LIN {X 0,Y 368.929,Z 1065.584,A -85,B 0,C 180,E1 16268.801,E2 16268.801} C_VEL
LIN {X 0,Y 361.367,Z 1080.301,A -85,B 0,C 180,E1 16265.652,E2 16265.652} C_VEL
LIN {X 0,Y 353.629,Z 1094.954,A -85,B 0,C 180,E1 16261.908,E2 16261.908} C_VEL
LIN {X 0,Y 348.28,Z 1105.205,A -85,B 0,C 180,E1 16258.82,E2 16258.82} C_VEL
LIN {X 0,Y 344.292,Z 1113.061,A -85,B 0,C 180,E1 16256.113,E2 16256.113} C_VEL
LIN {X 0,Y 341.847,Z 1116.356,A -85,B 0,C 180,E1 16255.008,E2 16255.008} C_VEL
LIN {X 0,Y 332.302,Z 1125.106,A -85,B 0,C 180,E1 16252.144,E2 16252.144} C_VEL
LIN {X 0,Y 330.487,Z 1127.448,A -85,B 0,C 180,E1 16251.111,E2 16251.111} C_VEL
LIN {X 0,Y 327.162,Z 1134.807,A -85,B 0,C 180,E1 16247.181,E2 16247.181} C_VEL
LIN {X 0,Y 324.967,Z 1140.258,A -85,B 0,C 180,E1 16243.693,E2 16243.693} C_VEL
LIN {X 0,Y 323.573,Z 1144.448,A -85,B 0,C 180,E1 16240.461,E2 16240.461} C_VEL
LIN {X 0,Y 322.533,Z 1148.193,A -85,B 0,C 180,E1 16236.887,E2 16236.887} C_VEL
LIN {X 0,Y 321.986,Z 1150.9,A -85,B 0,C 180,E1 16233.557,E2 16233.557} C_VEL
LIN {X 0,Y 321.773,Z 1152.88,A -85,B 0,C 180,E1 16230.226,E2 16230.226} C_VEL
LIN {X 0,Y 321.676,Z 1154.208,A -85,B 0,C 180,E1 16226.79,E2 16226.79} C_VEL
LIN {X 0,Y 321.778,Z 1154.811,A -85,B 0,C 180,E1 16223.438,E2 16223.438} C_VEL
LIN {X 0,Y 322.051,Z 1154.692,A -85,B 0,C 180,E1 16219.827,E2 16219.827} C_VEL
LIN {X 0,Y 322.549,Z 1153.785,A -85,B 0,C 180,E1 16216.2,E2 16216.2} C_VEL
LIN {X 0,Y 323.386,Z 1152.158,A -85,B 0,C 180,E1 16212.681,E2 16212.681} C_VEL
LIN {X 0,Y 324.964,Z 1149.492,A -85,B 0,C 180,E1 16208.85,E2 16208.85} C_VEL
LIN {X 0,Y 327.742,Z 1145.238,A -85,B 0,C 180,E1 16204.374,E2 16204.374} C_VEL
LIN {X 0,Y 332.024,Z 1139.047,A -85,B 0,C 180,E1 16199.655,E2 16199.655} C_VEL
LIN {X 0,Y 336.888,Z 1132.582,A -85,B 0,C 180,E1 16195.74,E2 16195.74} C_VEL
LIN {X 0,Y 344.034,Z 1123.589,A -85,B 0,C 180,E1 16191.307,E2 16191.307} C_VEL
LIN {X 0,Y 351.989,Z 1113.581,A -85,B 0,C 180,E1 16187.365,E2 16187.365} C_VEL
LIN {X 0,Y 361.723,Z 1101.762,A -85,B 0,C 180,E1 16183.458,E2 16183.458} C_VEL
LIN {X 0,Y 372.861,Z 1088.013,A -85,B 0,C 180,E1 16179.761,E2 16179.761} C_VEL
LIN {X 0,Y 385.536,Z 1072.73,A -85,B 0,C 180,E1 16176.297,E2 16176.297} C_VEL
LIN {X 0,Y 402.18,Z 1053.149,A -85,B 0,C 180,E1 16172.616,E2 16172.616} C_VEL
LIN {X 0,Y 414.234,Z 1039.577,A -85,B 0,C 180,E1 16170.456,E2 16170.456} C_VEL
LIN {X 0,Y 397.297,Z 1065.107,A -85,B 0,C 180,E1 16167.737,E2 16167.737} C_VEL
LIN {X 0,Y 379.335,Z 1097.703,A -85,B 0,C 180,E1 16163.762,E2 16163.762} C_VEL
LIN {X 0,Y 366.086,Z 1125.2,A -85,B 0,C 180,E1 16159.865,E2 16159.865} C_VEL
LIN {X 0,Y 355.502,Z 1148.51,A -85,B 0,C 180,E1 16155.995,E2 16155.995} C_VEL
LIN {X 0,Y 348.419,Z 1164.919,A -85,B 0,C 180,E1 16152.854,E2 16152.854} C_VEL
LIN {X 0,Y 342.515,Z 1179.307,A -85,B 0,C 180,E1 16149.74,E2 16149.74} C_VEL
LIN {X 0,Y 337.4,Z 1192.323,A -85,B 0,C 180,E1 16146.559,E2 16146.559} C_VEL
LIN {X 0,Y 333.277,Z 1203.483,A -85,B 0,C 180,E1 16143.483,E2 16143.483} C_VEL
LIN {X 0,Y 329.754,Z 1213.978,A -85,B 0,C 180,E1 16140.21,E2 16140.21} C_VEL
LIN {X 0,Y 326.806,Z 1223.77,A -85,B 0,C 180,E1 16136.728,E2 16136.728} C_VEL
LIN {X 0,Y 324.695,Z 1231.919,A -85,B 0,C 180,E1 16133.406,E2 16133.406} C_VEL
LIN {X 0,Y 323.147,Z 1239.311,A -85,B 0,C 180,E1 16129.899,E2 16129.899} C_VEL
LIN {X 0,Y 322.162,Z 1245.863,A -85,B 0,C 180,E1 16126.22,E2 16126.22} C_VEL
LIN {X 0,Y 321.683,Z 1251.131,A -85,B 0,C 180,E1 16122.567,E2 16122.567} C_VEL
LIN {X 0,Y 321.55,Z 1254.796,A -85,B 0,C 180,E1 16119.305,E2 16119.305} C_VEL
LIN {X 0,Y 321.644,Z 1257.645,A -85,B 0,C 180,E1 16115.855,E2 16115.855} C_VEL
LIN {X 0,Y 321.714,Z 1259.335,A -85,B 0,C 180,E1 16112.494,E2 16112.494} C_VEL
LIN {X 0,Y 321.649,Z 1259.923,A -85,B 0,C 180,E1 16109.109,E2 16109.109} C_VEL
LIN {X 0,Y 321.554,Z 1259.487,A -85,B 0,C 180,E1 16105.899,E2 16105.899} C_VEL
LIN {X 0,Y 321.358,Z 1257.951,A -85,B 0,C 180,E1 16102.491,E2 16102.491} C_VEL
LIN {X 0,Y 321.322,Z 1255.176,A -85,B 0,C 180,E1 16098.876,E2 16098.876} C_VEL
LIN {X 0,Y 321.576,Z 1251.22,A -85,B 0,C 180,E1 16095.229,E2 16095.229} C_VEL
LIN {X 0,Y 322.325,Z 1246.263,A -85,B 0,C 180,E1 16091.669,E2 16091.669} C_VEL
LIN {X 0,Y 323.717,Z 1240.102,A -85,B 0,C 180,E1 16088.054,E2 16088.054} C_VEL
LIN {X 0,Y 325.87,Z 1232.599,A -85,B 0,C 180,E1 16084.365,E2 16084.365} C_VEL
LIN {X 0,Y 329.419,Z 1222.452,A -85,B 0,C 180,E1 16080.146,E2 16080.146} C_VEL
LIN {X 0,Y 334.451,Z 1209.771,A -85,B 0,C 180,E1 16075.803,E2 16075.803} C_VEL
LIN {X 0,Y 339.559,Z 1198.071,A -85,B 0,C 180,E1 16072.384,E2 16072.384} C_VEL
LIN {X 0,Y 345.401,Z 1185.305,A -85,B 0,C 180,E1 16069.139,E2 16069.139} C_VEL
LIN {X 0,Y 353.389,Z 1168.407,A -85,B 0,C 180,E1 16065.437,E2 16065.437} C_VEL
LIN {X 0,Y 361.45,Z 1151.342,A -85,B 0,C 180,E1 16062.304,E2 16062.304} C_VEL
LIN {X 0,Y 369.122,Z 1135.016,A -85,B 0,C 180,E1 16059.709,E2 16059.709} C_VEL
LIN {X 0,Y 377.835,Z 1116.171,A -85,B 0,C 180,E1 16057.112,E2 16057.112} C_VEL
LIN {X 0,Y 387.715,Z 1093.832,A -85,B 0,C 180,E1 16054.517,E2 16054.517} C_VEL
LIN {X 0,Y 395.54,Z 1075.271,A -85,B 0,C 180,E1 16052.671,E2 16052.671} C_VEL
LIN {X 0,Y 403.455,Z 1055.515,A -85,B 0,C 180,E1 16050.964,E2 16050.964} C_VEL
LIN {X 0,Y 412.389,Z 1031.699,A -85,B 0,C 180,E1 16049.208,E2 16049.208} C_VEL
LIN {X 0,Y 420.728,Z 1007.097,A -85,B 0,C 180,E1 16047.716,E2 16047.716} C_VEL
LIN {X 0,Y 427.295,Z 986.002,A -85,B 0,C 180,E1 16046.634,E2 16046.634} C_VEL
LIN {X 0,Y 434.084,Z 962.064,A -85,B 0,C 180,E1 16045.606,E2 16045.606} C_VEL
LIN {X 0,Y 440.942,Z 933.969,A -85,B 0,C 180,E1 16044.644,E2 16044.644} C_VEL
LIN {X 0,Y 445.717,Z 910.846,A -85,B 0,C 180,E1 16044.015,E2 16044.015} C_VEL
LIN {X 0,Y 449.567,Z 887.226,A -85,B 0,C 180,E1 16043.462,E2 16043.462} C_VEL
LIN {X 0,Y 453.668,Z 850.311,A -85,B 0,C 180,E1 16042.756,E2 16042.756} C_VEL
LIN {X 0,Y 474.582,Z 637.863,A -85,B 0,C 180,E1 16039.052,E2 16039.052} C_VEL
LIN {X 0,Y 480.593,Z 579.148,A -85,B 0,C 180,E1 16038.031,E2 16038.031} C_VEL
LIN {X 0,Y 471.163,Z 563.283,A -85,B 0,C 180,E1 16034.942,E2 16034.942} C_VEL
LIN {X 0,Y 462.699,Z 549.888,A -85,B 0,C 180,E1 16031.878,E2 16031.878} C_VEL
LIN {X 0,Y 454.912,Z 537.8,A -85,B 0,C 180,E1 16028.723,E2 16028.723} C_VEL
LIN {X 0,Y 448.462,Z 528.192,A -85,B 0,C 180,E1 16025.822,E2 16025.822} C_VEL
LIN {X 0,Y 442.933,Z 519.88,A -85,B 0,C 180,E1 16023.041,E2 16023.041} C_VEL
LIN {X 0,Y 437.602,Z 512.312,A -85,B 0,C 180,E1 16020.065,E2 16020.065} C_VEL
LIN {X 0,Y 434.436,Z 507.764,A -85,B 0,C 180,E1 16018.087,E2 16018.087} C_VEL
LIN {X 0,Y 431.277,Z 503.161,A -85,B 0,C 180,E1 16015.945,E2 16015.945} C_VEL
LIN {X 0,Y 428.043,Z 498.552,A -85,B 0,C 180,E1 16013.562,E2 16013.562} C_VEL
LIN {X 0,Y 424.911,Z 493.865,A -85,B 0,C 180,E1 16010.929,E2 16010.929} C_VEL
LIN {X 0,Y 421.631,Z 489.288,A -85,B 0,C 180,E1 16007.815,E2 16007.815} C_VEL
LIN {X 0,Y 420.488,Z 487.518,A -85,B 0,C 180,E1 16006.546,E2 16006.546} C_VEL
LIN {X 0,Y 417.521,Z 483.166,A -85,B 0,C 180,E1 16002.868,E2 16002.868} C_VEL
LIN {X 0,Y 414.516,Z 480.784,A -85,B 0,C 180,E1 15998.787,E2 15998.787} C_VEL
LIN {X 0,Y 412.902,Z 477.95,A -85,B 0,C 180,E1 15995.385,E2 15995.385} C_VEL
LIN {X 0,Y 412.303,Z 476.965,A -85,B 0,C 180,E1 15993.653,E2 15993.653} C_VEL
LIN {X 0,Y 410.774,Z 476.217,A -85,B 0,C 180,E1 15989.095,E2 15989.095} C_VEL
LIN {X 0,Y 410.291,Z 475.897,A -85,B 0,C 180,E1 15985.212,E2 15985.212} C_VEL
LIN {X 0,Y 410.589,Z 476.045,A -85,B 0,C 180,E1 15980.531,E2 15980.531} C_VEL
LIN {X 0,Y 411.65,Z 476.625,A -85,B 0,C 180,E1 15976.371,E2 15976.371} C_VEL
LIN {X 0,Y 412.909,Z 477.464,A -85,B 0,C 180,E1 15973.408,E2 15973.408} C_VEL
LIN {X 0,Y 414.387,Z 480.345,A -85,B 0,C 180,E1 15970.29,E2 15970.29} C_VEL
LIN {X 0,Y 417.361,Z 482.989,A -85,B 0,C 180,E1 15966.281,E2 15966.281} C_VEL
LIN {X 0,Y 418.392,Z 483.769,A -85,B 0,C 180,E1 15965.166,E2 15965.166} C_VEL
LIN {X 0,Y 421.167,Z 487.9,A -85,B 0,C 180,E1 15962.126,E2 15962.126} C_VEL
LIN {X 0,Y 423.64,Z 489.996,A -85,B 0,C 180,E1 15959.979,E2 15959.979} C_VEL
LIN {X 0,Y 426.809,Z 494.304,A -85,B 0,C 180,E1 15957.39,E2 15957.39} C_VEL
LIN {X 0,Y 428.742,Z 496.203,A -85,B 0,C 180,E1 15956.05,E2 15956.05} C_VEL
LIN {X 0,Y 432.452,Z 500.769,A -85,B 0,C 180,E1 15953.578,E2 15953.578} C_VEL
LIN {X 0,Y 433.913,Z 502.443,A -85,B 0,C 180,E1 15952.704,E2 15952.704} C_VEL
LIN {X 0,Y 438.68,Z 508.376,A -85,B 0,C 180,E1 15949.992,E2 15949.992} C_VEL
LIN {X 0,Y 443.421,Z 514.255,A -85,B 0,C 180,E1 15947.587,E2 15947.587} C_VEL
LIN {X 0,Y 447.969,Z 520.088,A -85,B 0,C 180,E1 15945.47,E2 15945.47} C_VEL
LIN {X 0,Y 454.659,Z 528.643,A -85,B 0,C 180,E1 15942.669,E2 15942.669} C_VEL
LIN {X 0,Y 463.73,Z 540.901,A -85,B 0,C 180,E1 15939.272,E2 15939.272} C_VEL
LIN {X 0,Y 474.803,Z 556.321,A -85,B 0,C 180,E1 15935.65,E2 15935.65} C_VEL
LIN {X 0,Y 476.31,Z 558.799,A -85,B 0,C 180,E1 15935.176,E2 15935.176} C_VEL
LIN {X 0,Y 455.359,Z 771.033,A -85,B 0,C 180,E1 15931.537,E2 15931.537} C_VEL
LIN {X 0,Y 451.923,Z 800.539,A -85,B 0,C 180,E1 15930.948,E2 15930.948} C_VEL
LIN {X 0,Y 448.327,Z 824.07,A -85,B 0,C 180,E1 15930.335,E2 15930.335} C_VEL
LIN {X 0,Y 443.229,Z 851.426,A -85,B 0,C 180,E1 15929.441,E2 15929.441} C_VEL
LIN {X 0,Y 437.133,Z 877.659,A -85,B 0,C 180,E1 15928.362,E2 15928.362} C_VEL
LIN {X 0,Y 431.224,Z 899.891,A -85,B 0,C 180,E1 15927.276,E2 15927.276} C_VEL
LIN {X 0,Y 423.599,Z 925.285,A -85,B 0,C 180,E1 15925.804,E2 15925.804} C_VEL
LIN {X 0,Y 415.695,Z 948.263,A -85,B 0,C 180,E1 15924.202,E2 15924.202} C_VEL
LIN {X 0,Y 408.347,Z 967.91,A -85,B 0,C 180,E1 15922.613,E2 15922.613} C_VEL
LIN {X 0,Y 399.847,Z 988.995,A -85,B 0,C 180,E1 15920.646,E2 15920.646} C_VEL
LIN {X 0,Y 390.613,Z 1009.923,A -85,B 0,C 180,E1 15918.333,E2 15918.333} C_VEL
LIN {X 0,Y 382.76,Z 1026.711,A -85,B 0,C 180,E1 15916.179,E2 15916.179} C_VEL
LIN {X 0,Y 375.211,Z 1042.141,A -85,B 0,C 180,E1 15913.91,E2 15913.91} C_VEL
LIN {X 0,Y 366.367,Z 1059.568,A -85,B 0,C 180,E1 15910.943,E2 15910.943} C_VEL
LIN {X 0,Y 357.73,Z 1075.65,A -85,B 0,C 180,E1 15907.658,E2 15907.658} C_VEL
LIN {X 0,Y 351.471,Z 1087.232,A -85,B 0,C 180,E1 15904.92,E2 15904.92} C_VEL
LIN {X 0,Y 345.778,Z 1097.775,A -85,B 0,C 180,E1 15902.066,E2 15902.066} C_VEL
LIN {X 0,Y 340.542,Z 1107.574,A -85,B 0,C 180,E1 15899.022,E2 15899.022} C_VEL
LIN {X 0,Y 335.171,Z 1117.965,A -85,B 0,C 180,E1 15895.265,E2 15895.265} C_VEL
LIN {X 0,Y 330.487,Z 1127.448,A -85,B 0,C 180,E1 15891.111,E2 15891.111} C_VEL
LIN {X 0,Y 328.335,Z 1130.13,A -85,B 0,C 180,E1 15889.895,E2 15889.895} C_VEL
LIN {X 0,Y 319.625,Z 1137.342,A -85,B 0,C 180,E1 15886.708,E2 15886.708} C_VEL
LIN {X 0,Y 318.186,Z 1139.299,A -85,B 0,C 180,E1 15885.596,E2 15885.596} C_VEL
LIN {X 0,Y 315.874,Z 1145.454,A -85,B 0,C 180,E1 15880.939,E2 15880.939} C_VEL
LIN {X 0,Y 314.69,Z 1149.43,A -85,B 0,C 180,E1 15877.107,E2 15877.107} C_VEL
LIN {X 0,Y 314.104,Z 1152.208,A -85,B 0,C 180,E1 15873.635,E2 15873.635} C_VEL
LIN {X 0,Y 313.868,Z 1154.335,A -85,B 0,C 180,E1 15869.946,E2 15869.946} C_VEL
LIN {X 0,Y 313.814,Z 1155.654,A -85,B 0,C 180,E1 15866.289,E2 15866.289} C_VEL
LIN {X 0,Y 313.896,Z 1156.194,A -85,B 0,C 180,E1 15862.869,E2 15862.869} C_VEL
LIN {X 0,Y 314.211,Z 1156.067,A -85,B 0,C 180,E1 15859.52,E2 15859.52} C_VEL
LIN {X 0,Y 314.721,Z 1155.279,A -85,B 0,C 180,E1 15856.046,E2 15856.046} C_VEL
LIN {X 0,Y 315.619,Z 1153.729,A -85,B 0,C 180,E1 15852.441,E2 15852.441} C_VEL
LIN {X 0,Y 317.303,Z 1151.147,A -85,B 0,C 180,E1 15848.517,E2 15848.517} C_VEL
LIN {X 0,Y 320.404,Z 1146.822,A -85,B 0,C 180,E1 15843.758,E2 15843.758} C_VEL
LIN {X 0,Y 325.016,Z 1140.675,A -85,B 0,C 180,E1 15838.925,E2 15838.925} C_VEL
LIN {X 0,Y 329.914,Z 1134.617,A -85,B 0,C 180,E1 15835.132,E2 15835.132} C_VEL
LIN {X 0,Y 337.131,Z 1126.172,A -85,B 0,C 180,E1 15830.784,E2 15830.784} C_VEL
LIN {X 0,Y 346.132,Z 1115.586,A -85,B 0,C 180,E1 15826.468,E2 15826.468} C_VEL
LIN {X 0,Y 356.799,Z 1103.475,A -85,B 0,C 180,E1 15822.383,E2 15822.383} C_VEL
LIN {X 0,Y 369.506,Z 1088.903,A -85,B 0,C 180,E1 15818.406,E2 15818.406} C_VEL
LIN {X 0,Y 385.189,Z 1071.414,A -85,B 0,C 180,E1 15814.475,E2 15814.475} C_VEL
LIN {X 0,Y 403.975,Z 1051.52,A -85,B 0,C 180,E1 15810.817,E2 15810.817} C_VEL
LIN {X 0,Y 405.211,Z 1050.316,A -85,B 0,C 180,E1 15810.58,E2 15810.58} C_VEL
LIN {X 0,Y 388.9,Z 1073.655,A -85,B 0,C 180,E1 15807.903,E2 15807.903} C_VEL
LIN {X 0,Y 370.301,Z 1105.753,A -85,B 0,C 180,E1 15803.707,E2 15803.707} C_VEL
LIN {X 0,Y 356.333,Z 1133.003,A -85,B 0,C 180,E1 15799.502,E2 15799.502} C_VEL
LIN {X 0,Y 347.555,Z 1151.474,A -85,B 0,C 180,E1 15796.228,E2 15796.228} C_VEL
LIN {X 0,Y 338.548,Z 1171.684,A -85,B 0,C 180,E1 15792.1,E2 15792.1} C_VEL
LIN {X 0,Y 331.317,Z 1188.657,A -85,B 0,C 180,E1 15787.999,E2 15787.999} C_VEL
LIN {X 0,Y 326.407,Z 1201.226,A -85,B 0,C 180,E1 15784.509,E2 15784.509} C_VEL
LIN {X 0,Y 322.393,Z 1212.348,A -85,B 0,C 180,E1 15780.986,E2 15780.986} C_VEL
LIN {X 0,Y 319.408,Z 1221.709,A -85,B 0,C 180,E1 15777.6,E2 15777.6} C_VEL
LIN {X 0,Y 317.107,Z 1229.927,A -85,B 0,C 180,E1 15774.199,E2 15774.199} C_VEL
LIN {X 0,Y 315.464,Z 1237.137,A -85,B 0,C 180,E1 15770.766,E2 15770.766} C_VEL
LIN {X 0,Y 314.371,Z 1243.776,A -85,B 0,C 180,E1 15767.014,E2 15767.014} C_VEL
LIN {X 0,Y 313.812,Z 1248.981,A -85,B 0,C 180,E1 15763.45,E2 15763.45} C_VEL
LIN {X 0,Y 313.653,Z 1253.065,A -85,B 0,C 180,E1 15759.912,E2 15759.912} C_VEL
LIN {X 0,Y 313.722,Z 1256.017,A -85,B 0,C 180,E1 15756.405,E2 15756.405} C_VEL
LIN {X 0,Y 313.812,Z 1257.863,A -85,B 0,C 180,E1 15752.922,E2 15752.922} C_VEL
LIN {X 0,Y 313.765,Z 1258.592,A -85,B 0,C 180,E1 15749.452,E2 15749.452} C_VEL
LIN {X 0,Y 313.661,Z 1258.215,A -85,B 0,C 180,E1 15745.978,E2 15745.978} C_VEL
LIN {X 0,Y 313.449,Z 1256.724,A -85,B 0,C 180,E1 15742.485,E2 15742.485} C_VEL
LIN {X 0,Y 313.4,Z 1253.985,A -85,B 0,C 180,E1 15738.778,E2 15738.778} C_VEL
LIN {X 0,Y 313.669,Z 1250,A -85,B 0,C 180,E1 15734.991,E2 15734.991} C_VEL
LIN {X 0,Y 314.437,Z 1245.103,A -85,B 0,C 180,E1 15731.374,E2 15731.374} C_VEL
LIN {X 0,Y 315.9,Z 1238.976,A -85,B 0,C 180,E1 15727.677,E2 15727.677} C_VEL
LIN {X 0,Y 318.151,Z 1231.476,A -85,B 0,C 180,E1 15723.897,E2 15723.897} C_VEL
LIN {X 0,Y 321.687,Z 1221.773,A -85,B 0,C 180,E1 15719.766,E2 15719.766} C_VEL
LIN {X 0,Y 327.14,Z 1208.628,A -85,B 0,C 180,E1 15715.142,E2 15715.142} C_VEL
LIN {X 0,Y 332.371,Z 1197.106,A -85,B 0,C 180,E1 15711.705,E2 15711.705} C_VEL
LIN {X 0,Y 338.183,Z 1184.869,A -85,B 0,C 180,E1 15708.526,E2 15708.526} C_VEL
LIN {X 0,Y 345.619,Z 1169.609,A -85,B 0,C 180,E1 15705.098,E2 15705.098} C_VEL
LIN {X 0,Y 354.896,Z 1150.65,A -85,B 0,C 180,E1 15701.525,E2 15701.525} C_VEL
LIN {X 0,Y 362.637,Z 1134.7,A -85,B 0,C 180,E1 15698.951,E2 15698.951} C_VEL
LIN {X 0,Y 370.83,Z 1117.486,A -85,B 0,C 180,E1 15696.534,E2 15696.534} C_VEL
LIN {X 0,Y 381.394,Z 1094.469,A -85,B 0,C 180,E1 15693.793,E2 15693.793} C_VEL
LIN {X 0,Y 389.993,Z 1074.531,A -85,B 0,C 180,E1 15691.798,E2 15691.798} C_VEL
LIN {X 0,Y 397.776,Z 1055.519,A -85,B 0,C 180,E1 15690.151,E2 15690.151} C_VEL
LIN {X 0,Y 406.896,Z 1031.853,A -85,B 0,C 180,E1 15688.391,E2 15688.391} C_VEL
LIN {X 0,Y 415.538,Z 1007.032,A -85,B 0,C 180,E1 15686.876,E2 15686.876} C_VEL
LIN {X 0,Y 422.443,Z 985.37,A -85,B 0,C 180,E1 15685.763,E2 15685.763} C_VEL
LIN {X 0,Y 429.36,Z 961.523,A -85,B 0,C 180,E1 15684.74,E2 15684.74} C_VEL
LIN {X 0,Y 436.385,Z 933.409,A -85,B 0,C 180,E1 15683.78,E2 15683.78} C_VEL
LIN {X 0,Y 441.272,Z 910.236,A -85,B 0,C 180,E1 15683.149,E2 15683.149} C_VEL
LIN {X 0,Y 445.234,Z 886.47,A -85,B 0,C 180,E1 15682.592,E2 15682.592} C_VEL
LIN {X 0,Y 449.401,Z 849.977,A -85,B 0,C 180,E1 15681.892,E2 15681.892} C_VEL
LIN {X 0,Y 470.846,Z 638.55,A -85,B 0,C 180,E1 15678.199,E2 15678.199} C_VEL
LIN {X 0,Y 476.609,Z 583.778,A -85,B 0,C 180,E1 15677.247,E2 15677.247} C_VEL
LIN {X 0,Y 467.496,Z 568.387,A -85,B 0,C 180,E1 15674.176,E2 15674.176} C_VEL
LIN {X 0,Y 458.486,Z 554.028,A -85,B 0,C 180,E1 15670.81,E2 15670.81} C_VEL
LIN {X 0,Y 450.098,Z 541.072,A -85,B 0,C 180,E1 15667.275,E2 15667.275} C_VEL
LIN {X 0,Y 442.156,Z 529.252,A -85,B 0,C 180,E1 15663.436,E2 15663.436} C_VEL
LIN {X 0,Y 436.099,Z 520.425,A -85,B 0,C 180,E1 15660.066,E2 15660.066} C_VEL
LIN {X 0,Y 432.802,Z 515.672,A -85,B 0,C 180,E1 15658.014,E2 15658.014} C_VEL
LIN {X 0,Y 429.487,Z 510.786,A -85,B 0,C 180,E1 15655.727,E2 15655.727} C_VEL
LIN {X 0,Y 426.243,Z 506.171,A -85,B 0,C 180,E1 15653.332,E2 15653.332} C_VEL
LIN {X 0,Y 422.555,Z 500.812,A -85,B 0,C 180,E1 15650.19,E2 15650.19} C_VEL
LIN {X 0,Y 419.553,Z 496.204,A -85,B 0,C 180,E1 15647.195,E2 15647.195} C_VEL
LIN {X 0,Y 416.221,Z 491.264,A -85,B 0,C 180,E1 15643.173,E2 15643.173} C_VEL
LIN {X 0,Y 412.967,Z 488.655,A -85,B 0,C 180,E1 15638.774,E2 15638.774} C_VEL
LIN {X 0,Y 411.35,Z 485.853,A -85,B 0,C 180,E1 15635.38,E2 15635.38} C_VEL
LIN {X 0,Y 410.779,Z 484.846,A -85,B 0,C 180,E1 15633.704,E2 15633.704} C_VEL
LIN {X 0,Y 409.241,Z 484.068,A -85,B 0,C 180,E1 15629.13,E2 15629.13} C_VEL
LIN {X 0,Y 408.756,Z 483.742,A -85,B 0,C 180,E1 15625.031,E2 15625.031} C_VEL
LIN {X 0,Y 409.103,Z 483.934,A -85,B 0,C 180,E1 15620.181,E2 15620.181} C_VEL
LIN {X 0,Y 410.296,Z 484.537,A -85,B 0,C 180,E1 15615.964,E2 15615.964} C_VEL
LIN {X 0,Y 411.403,Z 485.379,A -85,B 0,C 180,E1 15613.389,E2 15613.389} C_VEL
LIN {X 0,Y 412.891,Z 488.246,A -85,B 0,C 180,E1 15610.284,E2 15610.284} C_VEL
LIN {X 0,Y 415.9,Z 490.867,A -85,B 0,C 180,E1 15606.257,E2 15606.257} C_VEL
LIN {X 0,Y 416.777,Z 491.537,A -85,B 0,C 180,E1 15605.322,E2 15605.322} C_VEL
LIN {X 0,Y 419.596,Z 495.713,A -85,B 0,C 180,E1 15602.225,E2 15602.225} C_VEL
LIN {X 0,Y 421.985,Z 497.776,A -85,B 0,C 180,E1 15600.132,E2 15600.132} C_VEL
LIN {X 0,Y 425.149,Z 502.046,A -85,B 0,C 180,E1 15597.544,E2 15597.544} C_VEL
LIN {X 0,Y 426.986,Z 503.883,A -85,B 0,C 180,E1 15596.247,E2 15596.247} C_VEL
LIN {X 0,Y 430.86,Z 508.591,A -85,B 0,C 180,E1 15593.67,E2 15593.67} C_VEL
LIN {X 0,Y 432.817,Z 511.133,A -85,B 0,C 180,E1 15592.47,E2 15592.47} C_VEL
LIN {X 0,Y 436.834,Z 516.009,A -85,B 0,C 180,E1 15590.203,E2 15590.203} C_VEL
LIN {X 0,Y 441.502,Z 521.861,A -85,B 0,C 180,E1 15587.802,E2 15587.802} C_VEL
LIN {X 0,Y 445.909,Z 527.519,A -85,B 0,C 180,E1 15585.743,E2 15585.743} C_VEL
LIN {X 0,Y 452.569,Z 536.118,A -85,B 0,C 180,E1 15582.927,E2 15582.927} C_VEL
LIN {X 0,Y 461.897,Z 548.801,A -85,B 0,C 180,E1 15579.406,E2 15579.406} C_VEL
LIN {X 0,Y 472.306,Z 563.557,A -85,B 0,C 180,E1 15575.968,E2 15575.968} C_VEL
LIN {X 0,Y 451.01,Z 773.161,A -85,B 0,C 180,E1 15572.369,E2 15572.369} C_VEL
LIN {X 0,Y 447.547,Z 801.925,A -85,B 0,C 180,E1 15571.788,E2 15571.788} C_VEL
LIN {X 0,Y 443.789,Z 825.809,A -85,B 0,C 180,E1 15571.162,E2 15571.162} C_VEL
LIN {X 0,Y 438.534,Z 853.134,A -85,B 0,C 180,E1 15570.261,E2 15570.261} C_VEL
LIN {X 0,Y 432.45,Z 878.743,A -85,B 0,C 180,E1 15569.205,E2 15569.205} C_VEL
LIN {X 0,Y 426.623,Z 900.22,A -85,B 0,C 180,E1 15568.157,E2 15568.157} C_VEL
LIN {X 0,Y 419.015,Z 925.265,A -85,B 0,C 180,E1 15566.717,E2 15566.717} C_VEL
LIN {X 0,Y 410.725,Z 949.006,A -85,B 0,C 180,E1 15565.07,E2 15565.07} C_VEL
LIN {X 0,Y 403.519,Z 967.99,A -85,B 0,C 180,E1 15563.542,E2 15563.542} C_VEL
LIN {X 0,Y 395.773,Z 986.821,A -85,B 0,C 180,E1 15561.801,E2 15561.801} C_VEL
LIN {X 0,Y 385.631,Z 1009.597,A -85,B 0,C 180,E1 15559.328,E2 15559.328} C_VEL
LIN {X 0,Y 377.432,Z 1026.716,A -85,B 0,C 180,E1 15557.138,E2 15557.138} C_VEL
LIN {X 0,Y 369.99,Z 1041.565,A -85,B 0,C 180,E1 15554.964,E2 15554.964} C_VEL
LIN {X 0,Y 362.586,Z 1055.798,A -85,B 0,C 180,E1 15552.584,E2 15552.584} C_VEL
LIN {X 0,Y 354.041,Z 1071.787,A -85,B 0,C 180,E1 15549.501,E2 15549.501} C_VEL
LIN {X 0,Y 345.717,Z 1086.701,A -85,B 0,C 180,E1 15546.057,E2 15546.057} C_VEL
LIN {X 0,Y 339.194,Z 1098.336,A -85,B 0,C 180,E1 15542.905,E2 15542.905} C_VEL
LIN {X 0,Y 333.644,Z 1108.338,A -85,B 0,C 180,E1 15539.77,E2 15539.77} C_VEL
LIN {X 0,Y 328.602,Z 1117.682,A -85,B 0,C 180,E1 15536.373,E2 15536.373} C_VEL
LIN {X 0,Y 323.461,Z 1127.792,A -85,B 0,C 180,E1 15532.024,E2 15532.024} C_VEL
LIN {X 0,Y 319.552,Z 1135.994,A -85,B 0,C 180,E1 15527.6,E2 15527.6} C_VEL
LIN {X 0,Y 318.186,Z 1139.299,A -85,B 0,C 180,E1 15525.596,E2 15525.596} C_VEL
LIN {X 0,Y 316.46,Z 1141.488,A -85,B 0,C 180,E1 15524.288,E2 15524.288} C_VEL
LIN {X 0,Y 308.48,Z 1147.125,A -85,B 0,C 180,E1 15520.703,E2 15520.703} C_VEL
LIN {X 0,Y 307.474,Z 1148.466,A -85,B 0,C 180,E1 15519.606,E2 15519.606} C_VEL
LIN {X 0,Y 306.366,Z 1152.909,A -85,B 0,C 180,E1 15514.603,E2 15514.603} C_VEL
LIN {X 0,Y 305.994,Z 1155.436,A -85,B 0,C 180,E1 15510.384,E2 15510.384} C_VEL
LIN {X 0,Y 305.894,Z 1156.833,A -85,B 0,C 180,E1 15506.814,E2 15506.814} C_VEL
LIN {X 0,Y 306.007,Z 1157.523,A -85,B 0,C 180,E1 15503.289,E2 15503.289} C_VEL
LIN {X 0,Y 306.349,Z 1157.503,A -85,B 0,C 180,E1 15499.446,E2 15499.446} C_VEL
LIN {X 0,Y 306.937,Z 1156.717,A -85,B 0,C 180,E1 15495.687,E2 15495.687} C_VEL
LIN {X 0,Y 307.926,Z 1155.208,A -85,B 0,C 180,E1 15491.995,E2 15491.995} C_VEL
LIN {X 0,Y 309.758,Z 1152.68,A -85,B 0,C 180,E1 15487.979,E2 15487.979} C_VEL
LIN {X 0,Y 312.949,Z 1148.595,A -85,B 0,C 180,E1 15483.297,E2 15483.297} C_VEL
LIN {X 0,Y 317.819,Z 1142.644,A -85,B 0,C 180,E1 15478.377,E2 15478.377} C_VEL
LIN {X 0,Y 323.003,Z 1136.697,A -85,B 0,C 180,E1 15474.493,E2 15474.493} C_VEL
LIN {X 0,Y 330.907,Z 1128.076,A -85,B 0,C 180,E1 15469.906,E2 15469.906} C_VEL
LIN {X 0,Y 340.396,Z 1117.68,A -85,B 0,C 180,E1 15465.541,E2 15465.541} C_VEL
LIN {X 0,Y 351.623,Z 1105.82,A -85,B 0,C 180,E1 15461.428,E2 15461.428} C_VEL
LIN {X 0,Y 367.044,Z 1089.549,A -85,B 0,C 180,E1 15456.903,E2 15456.903} C_VEL
LIN {X 0,Y 386.297,Z 1070.059,A -85,B 0,C 180,E1 15452.565,E2 15452.565} C_VEL
LIN {X 0,Y 396.221,Z 1060.536,A -85,B 0,C 180,E1 15450.719,E2 15450.719} C_VEL
LIN {X 0,Y 382.479,Z 1078.959,A -85,B 0,C 180,E1 15448.455,E2 15448.455} C_VEL
LIN {X 0,Y 364.569,Z 1107.301,A -85,B 0,C 180,E1 15444.544,E2 15444.544} C_VEL
LIN {X 0,Y 350.708,Z 1132.504,A -85,B 0,C 180,E1 15440.521,E2 15440.521} C_VEL
LIN {X 0,Y 339.116,Z 1155.538,A -85,B 0,C 180,E1 15436.251,E2 15436.251} C_VEL
LIN {X 0,Y 330.718,Z 1173.259,A -85,B 0,C 180,E1 15432.392,E2 15432.392} C_VEL
LIN {X 0,Y 324.523,Z 1187.118,A -85,B 0,C 180,E1 15428.942,E2 15428.942} C_VEL
LIN {X 0,Y 319.357,Z 1199.619,A -85,B 0,C 180,E1 15425.395,E2 15425.395} C_VEL
LIN {X 0,Y 315.086,Z 1210.775,A -85,B 0,C 180,E1 15421.788,E2 15421.788} C_VEL
LIN {X 0,Y 311.879,Z 1220.154,A -85,B 0,C 180,E1 15418.326,E2 15418.326} C_VEL
LIN {X 0,Y 309.4,Z 1228.588,A -85,B 0,C 180,E1 15414.754,E2 15414.754} C_VEL
LIN {X 0,Y 307.622,Z 1235.928,A -85,B 0,C 180,E1 15411.148,E2 15411.148} C_VEL
LIN {X 0,Y 306.53,Z 1242.012,A -85,B 0,C 180,E1 15407.659,E2 15407.659} C_VEL
LIN {X 0,Y 305.924,Z 1247.047,A -85,B 0,C 180,E1 15404.189,E2 15404.189} C_VEL
LIN {X 0,Y 305.745,Z 1251.287,A -85,B 0,C 180,E1 15400.552,E2 15400.552} C_VEL
LIN {X 0,Y 305.801,Z 1254.53,A -85,B 0,C 180,E1 15396.76,E2 15396.76} C_VEL
LIN {X 0,Y 305.909,Z 1256.465,A -85,B 0,C 180,E1 15393.185,E2 15393.185} C_VEL
LIN {X 0,Y 305.885,Z 1257.258,A -85,B 0,C 180,E1 15389.625,E2 15389.625} C_VEL
LIN {X 0,Y 305.771,Z 1256.934,A -85,B 0,C 180,E1 15386.062,E2 15386.062} C_VEL
LIN {X 0,Y 305.541,Z 1255.489,A -85,B 0,C 180,E1 15382.478,E2 15382.478} C_VEL
LIN {X 0,Y 305.479,Z 1252.786,A -85,B 0,C 180,E1 15378.674,E2 15378.674} C_VEL
LIN {X 0,Y 305.769,Z 1248.755,A -85,B 0,C 180,E1 15374.727,E2 15374.727} C_VEL
LIN {X 0,Y 306.593,Z 1243.783,A -85,B 0,C 180,E1 15370.966,E2 15370.966} C_VEL
LIN {X 0,Y 308.191,Z 1237.476,A -85,B 0,C 180,E1 15367.088,E2 15367.088} C_VEL
LIN {X 0,Y 310.745,Z 1229.518,A -85,B 0,C 180,E1 15363.019,E2 15363.019} C_VEL
LIN {X 0,Y 315.173,Z 1218.19,A -85,B 0,C 180,E1 15358.222,E2 15358.222} C_VEL
LIN {X 0,Y 320.412,Z 1206.324,A -85,B 0,C 180,E1 15354.079,E2 15354.079} C_VEL
LIN {X 0,Y 325.928,Z 1194.62,A -85,B 0,C 180,E1 15350.578,E2 15350.578} C_VEL
LIN {X 0,Y 332.819,Z 1180.765,A -85,B 0,C 180,E1 15347.002,E2 15347.002} C_VEL
LIN {X 0,Y 341.633,Z 1163.335,A -85,B 0,C 180,E1 15343.217,E2 15343.217} C_VEL
LIN {X 0,Y 349.444,Z 1147.879,A -85,B 0,C 180,E1 15340.357,E2 15340.357} C_VEL
LIN {X 0,Y 357.185,Z 1132.428,A -85,B 0,C 180,E1 15337.87,E2 15337.87} C_VEL
LIN {X 0,Y 367.002,Z 1112.363,A -85,B 0,C 180,E1 15335.09,E2 15335.09} C_VEL
LIN {X 0,Y 377.097,Z 1090.464,A -85,B 0,C 180,E1 15332.566,E2 15332.566} C_VEL
LIN {X 0,Y 385.439,Z 1071.582,A -85,B 0,C 180,E1 15330.703,E2 15330.703} C_VEL
LIN {X 0,Y 394.395,Z 1050.169,A -85,B 0,C 180,E1 15328.885,E2 15328.885} C_VEL
LIN {X 0,Y 404.14,Z 1024.704,A -85,B 0,C 180,E1 15327.08,E2 15327.08} C_VEL
LIN {X 0,Y 411.516,Z 1003.79,A -85,B 0,C 180,E1 15325.841,E2 15325.841} C_VEL
LIN {X 0,Y 418.681,Z 981.616,A -85,B 0,C 180,E1 15324.725,E2 15324.725} C_VEL
LIN {X 0,Y 426.994,Z 952.593,A -85,B 0,C 180,E1 15323.543,E2 15323.543} C_VEL
LIN {X 0,Y 432.79,Z 929.081,A -85,B 0,C 180,E1 15322.787,E2 15322.787} C_VEL
LIN {X 0,Y 437.81,Z 905.019,A -85,B 0,C 180,E1 15322.15,E2 15322.15} C_VEL
LIN {X 0,Y 442.557,Z 874.082,A -85,B 0,C 180,E1 15321.464,E2 15321.464} C_VEL
LIN {X 0,Y 461.42,Z 691.94,A -85,B 0,C 180,E1 15318.25,E2 15318.25} C_VEL
LIN {X 0,Y 472.577,Z 588.422,A -85,B 0,C 180,E1 15316.47,E2 15316.47} C_VEL
LIN {X 0,Y 463.949,Z 573.965,A -85,B 0,C 180,E1 15313.491,E2 15313.491} C_VEL
LIN {X 0,Y 456.183,Z 561.32,A -85,B 0,C 180,E1 15310.514,E2 15310.514} C_VEL
LIN {X 0,Y 448.767,Z 549.792,A -85,B 0,C 180,E1 15307.361,E2 15307.361} C_VEL
LIN {X 0,Y 441.797,Z 539.109,A -85,B 0,C 180,E1 15304.023,E2 15304.023} C_VEL
LIN {X 0,Y 434.935,Z 528.964,A -85,B 0,C 180,E1 15300.263,E2 15300.263} C_VEL
LIN {X 0,Y 430.846,Z 523.157,A -85,B 0,C 180,E1 15297.739,E2 15297.739} C_VEL
LIN {X 0,Y 427.594,Z 518.28,A -85,B 0,C 180,E1 15295.44,E2 15295.44} C_VEL
LIN {X 0,Y 424.364,Z 513.687,A -85,B 0,C 180,E1 15293.03,E2 15293.03} C_VEL
LIN {X 0,Y 420.853,Z 508.521,A -85,B 0,C 180,E1 15290.012,E2 15290.012} C_VEL
LIN {X 0,Y 417.351,Z 503.202,A -85,B 0,C 180,E1 15286.421,E2 15286.421} C_VEL
LIN {X 0,Y 414.337,Z 498.82,A -85,B 0,C 180,E1 15282.733,E2 15282.733} C_VEL
LIN {X 0,Y 411.423,Z 496.533,A -85,B 0,C 180,E1 15278.769,E2 15278.769} C_VEL
LIN {X 0,Y 409.844,Z 493.872,A -85,B 0,C 180,E1 15275.496,E2 15275.496} C_VEL
LIN {X 0,Y 409.302,Z 492.783,A -85,B 0,C 180,E1 15273.914,E2 15273.914} C_VEL
LIN {X 0,Y 407.752,Z 491.928,A -85,B 0,C 180,E1 15269.332,E2 15269.332} C_VEL
LIN {X 0,Y 407.214,Z 491.601,A -85,B 0,C 180,E1 15265.273,E2 15265.273} C_VEL
LIN {X 0,Y 407.532,Z 491.75,A -85,B 0,C 180,E1 15260.545,E2 15260.545} C_VEL
LIN {X 0,Y 408.689,Z 492.363,A -85,B 0,C 180,E1 15256.181,E2 15256.181} C_VEL
LIN {X 0,Y 409.857,Z 493.216,A -85,B 0,C 180,E1 15253.469,E2 15253.469} C_VEL
LIN {X 0,Y 411.407,Z 496.166,A -85,B 0,C 180,E1 15250.257,E2 15250.257} C_VEL
LIN {X 0,Y 414.567,Z 498.807,A -85,B 0,C 180,E1 15246.1,E2 15246.1} C_VEL
LIN {X 0,Y 415.292,Z 499.611,A -85,B 0,C 180,E1 15245.293,E2 15245.293} C_VEL
LIN {X 0,Y 418.309,Z 503.801,A -85,B 0,C 180,E1 15242.049,E2 15242.049} C_VEL
LIN {X 0,Y 420.335,Z 505.556,A -85,B 0,C 180,E1 15240.285,E2 15240.285} C_VEL
LIN {X 0,Y 423.473,Z 509.79,A -85,B 0,C 180,E1 15237.694,E2 15237.694} C_VEL
LIN {X 0,Y 425.324,Z 511.708,A -85,B 0,C 180,E1 15236.379,E2 15236.379} C_VEL
LIN {X 0,Y 429.389,Z 516.516,A -85,B 0,C 180,E1 15233.691,E2 15233.691} C_VEL
LIN {X 0,Y 435.046,Z 523.734,A -85,B 0,C 180,E1 15230.377,E2 15230.377} C_VEL
LIN {X 0,Y 439.665,Z 529.567,A -85,B 0,C 180,E1 15227.982,E2 15227.982} C_VEL
LIN {X 0,Y 444.028,Z 535.182,A -85,B 0,C 180,E1 15225.94,E2 15225.94} C_VEL
LIN {X 0,Y 450.563,Z 543.745,A -85,B 0,C 180,E1 15223.141,E2 15223.141} C_VEL
LIN {X 0,Y 460.077,Z 556.699,A -85,B 0,C 180,E1 15219.539,E2 15219.539} C_VEL
LIN {X 0,Y 468.261,Z 568.615,A -85,B 0,C 180,E1 15216.762,E2 15216.762} C_VEL
LIN {X 0,Y 445.063,Z 789.887,A -85,B 0,C 180,E1 15212.938,E2 15212.938} C_VEL
LIN {X 0,Y 440.646,Z 820.153,A -85,B 0,C 180,E1 15212.215,E2 15212.215} C_VEL
LIN {X 0,Y 436.175,Z 844.001,A -85,B 0,C 180,E1 15211.48,E2 15211.48} C_VEL
LIN {X 0,Y 430.87,Z 867.913,A -85,B 0,C 180,E1 15210.584,E2 15210.584} C_VEL
LIN {X 0,Y 423.426,Z 896.107,A -85,B 0,C 180,E1 15209.286,E2 15209.286} C_VEL
LIN {X 0,Y 417.175,Z 916.806,A -85,B 0,C 180,E1 15208.145,E2 15208.145} C_VEL
LIN {X 0,Y 410.561,Z 936.555,A -85,B 0,C 180,E1 15206.892,E2 15206.892} C_VEL
LIN {X 0,Y 401.896,Z 960.196,A -85,B 0,C 180,E1 15205.148,E2 15205.148} C_VEL
LIN {X 0,Y 392.734,Z 982.426,A -85,B 0,C 180,E1 15203.185,E2 15203.185} C_VEL
LIN {X 0,Y 384.706,Z 1000.577,A -85,B 0,C 180,E1 15201.33,E2 15201.33} C_VEL
LIN {X 0,Y 376.251,Z 1018.571,A -85,B 0,C 180,E1 15199.21,E2 15199.21} C_VEL
LIN {X 0,Y 365.986,Z 1038.937,A -85,B 0,C 180,E1 15196.37,E2 15196.37} C_VEL
LIN {X 0,Y 357.989,Z 1053.963,A -85,B 0,C 180,E1 15193.909,E2 15193.909} C_VEL
LIN {X 0,Y 350.418,Z 1067.713,A -85,B 0,C 180,E1 15191.324,E2 15191.324} C_VEL
LIN {X 0,Y 343.463,Z 1080.058,A -85,B 0,C 180,E1 15188.661,E2 15188.661} C_VEL
LIN {X 0,Y 336.23,Z 1092.744,A -85,B 0,C 180,E1 15185.505,E2 15185.505} C_VEL
LIN {X 0,Y 328.177,Z 1106.782,A -85,B 0,C 180,E1 15181.34,E2 15181.34} C_VEL
LIN {X 0,Y 322.503,Z 1116.775,A -85,B 0,C 180,E1 15177.774,E2 15177.774} C_VEL
LIN {X 0,Y 317.9,Z 1125.225,A -85,B 0,C 180,E1 15174.242,E2 15174.242} C_VEL
LIN {X 0,Y 314.142,Z 1132.519,A -85,B 0,C 180,E1 15170.665,E2 15170.665} C_VEL
LIN {X 0,Y 310.916,Z 1139.451,A -85,B 0,C 180,E1 15166.62,E2 15166.62} C_VEL
LIN {X 0,Y 308.178,Z 1146.418,A -85,B 0,C 180,E1 15161.444,E2 15161.444} C_VEL
LIN {X 0,Y 307.474,Z 1148.466,A -85,B 0,C 180,E1 15159.606,E2 15159.606} C_VEL
LIN {X 0,Y 306.089,Z 1150.112,A -85,B 0,C 180,E1 15158.213,E2 15158.213} C_VEL
LIN {X 0,Y 299.025,Z 1154.321,A -85,B 0,C 180,E1 15154.374,E2 15154.374} C_VEL
LIN {X 0,Y 298.286,Z 1155.166,A -85,B 0,C 180,E1 15153.217,E2 15153.217} C_VEL
LIN {X 0,Y 298.057,Z 1157.26,A -85,B 0,C 180,E1 15149.284,E2 15149.284} C_VEL
LIN {X 0,Y 298.073,Z 1158.696,A -85,B 0,C 180,E1 15144.792,E2 15144.792} C_VEL
LIN {X 0,Y 298.417,Z 1159.018,A -85,B 0,C 180,E1 15139.985,E2 15139.985} C_VEL
LIN {X 0,Y 299.085,Z 1158.281,A -85,B 0,C 180,E1 15135.674,E2 15135.674} C_VEL
LIN {X 0,Y 300.195,Z 1156.795,A -85,B 0,C 180,E1 15131.695,E2 15131.695} C_VEL
LIN {X 0,Y 302.136,Z 1154.374,A -85,B 0,C 180,E1 15127.607,E2 15127.607} C_VEL
LIN {X 0,Y 305.524,Z 1150.411,A -85,B 0,C 180,E1 15122.814,E2 15122.814} C_VEL
LIN {X 0,Y 310.907,Z 1144.386,A -85,B 0,C 180,E1 15117.604,E2 15117.604} C_VEL
LIN {X 0,Y 316.979,Z 1137.958,A -85,B 0,C 180,E1 15113.297,E2 15113.297} C_VEL
LIN {X 0,Y 325.802,Z 1128.991,A -85,B 0,C 180,E1 15108.493,E2 15108.493} C_VEL
LIN {X 0,Y 335.6,Z 1119.06,A -85,B 0,C 180,E1 15104.269,E2 15104.269} C_VEL
LIN {X 0,Y 347.991,Z 1106.841,A -85,B 0,C 180,E1 15100.006,E2 15100.006} C_VEL
LIN {X 0,Y 364.453,Z 1090.961,A -85,B 0,C 180,E1 15095.526,E2 15095.526} C_VEL
LIN {X 0,Y 384.293,Z 1072.661,A -85,B 0,C 180,E1 15091.396,E2 15091.396} C_VEL
LIN {X 0,Y 387.062,Z 1070.146,A -85,B 0,C 180,E1 15090.863,E2 15090.863} C_VEL
LIN {X 0,Y 369.707,Z 1092.938,A -85,B 0,C 180,E1 15087.805,E2 15087.805} C_VEL
LIN {X 0,Y 350.039,Z 1123.806,A -85,B 0,C 180,E1 15083.028,E2 15083.028} C_VEL
LIN {X 0,Y 335.868,Z 1149.438,A -85,B 0,C 180,E1 15078.35,E2 15078.35} C_VEL
LIN {X 0,Y 325.107,Z 1170.411,A -85,B 0,C 180,E1 15073.788,E2 15073.788} C_VEL
LIN {X 0,Y 318.16,Z 1184.977,A -85,B 0,C 180,E1 15070.109,E2 15070.109} C_VEL
LIN {X 0,Y 312.77,Z 1197.055,A -85,B 0,C 180,E1 15066.638,E2 15066.638} C_VEL
LIN {X 0,Y 308.263,Z 1208.125,A -85,B 0,C 180,E1 15063.019,E2 15063.019} C_VEL
LIN {X 0,Y 304.742,Z 1217.629,A -85,B 0,C 180,E1 15059.482,E2 15059.482} C_VEL
LIN {X 0,Y 301.938,Z 1226.463,A -85,B 0,C 180,E1 15055.709,E2 15055.709} C_VEL
LIN {X 0,Y 299.954,Z 1234.093,A -85,B 0,C 180,E1 15051.922,E2 15051.922} C_VEL
LIN {X 0,Y 298.713,Z 1240.231,A -85,B 0,C 180,E1 15048.339,E2 15048.339} C_VEL
LIN {X 0,Y 298.027,Z 1245.624,A -85,B 0,C 180,E1 15044.574,E2 15044.574} C_VEL
LIN {X 0,Y 297.825,Z 1249.874,A -85,B 0,C 180,E1 15040.836,E2 15040.836} C_VEL
LIN {X 0,Y 297.869,Z 1253.02,A -85,B 0,C 180,E1 15037.134,E2 15037.134} C_VEL
LIN {X 0,Y 298.01,Z 1255.041,A -85,B 0,C 180,E1 15033.462,E2 15033.462} C_VEL
LIN {X 0,Y 298.008,Z 1255.914,A -85,B 0,C 180,E1 15029.808,E2 15029.808} C_VEL
LIN {X 0,Y 297.881,Z 1255.648,A -85,B 0,C 180,E1 15026.151,E2 15026.151} C_VEL
LIN {X 0,Y 297.63,Z 1254.165,A -85,B 0,C 180,E1 15022.333,E2 15022.333} C_VEL
LIN {X 0,Y 297.566,Z 1251.401,A -85,B 0,C 180,E1 15018.369,E2 15018.369} C_VEL
LIN {X 0,Y 297.88,Z 1247.464,A -85,B 0,C 180,E1 15014.423,E2 15014.423} C_VEL
LIN {X 0,Y 298.794,Z 1242.32,A -85,B 0,C 180,E1 15010.45,E2 15010.45} C_VEL
LIN {X 0,Y 300.602,Z 1235.617,A -85,B 0,C 180,E1 15006.267,E2 15006.267} C_VEL
LIN {X 0,Y 303.936,Z 1226.222,A -85,B 0,C 180,E1 15001.448,E2 15001.448} C_VEL
LIN {X 0,Y 308.627,Z 1214.933,A -85,B 0,C 180,E1 14996.803,E2 14996.803} C_VEL
LIN {X 0,Y 313.471,Z 1204.516,A -85,B 0,C 180,E1 14993.154,E2 14993.154} C_VEL
LIN {X 0,Y 319.402,Z 1192.516,A -85,B 0,C 180,E1 14989.527,E2 14989.527} C_VEL
LIN {X 0,Y 327.703,Z 1176.553,A -85,B 0,C 180,E1 14985.431,E2 14985.431} C_VEL
LIN {X 0,Y 335.943,Z 1160.749,A -85,B 0,C 180,E1 14982.043,E2 14982.043} C_VEL
LIN {X 0,Y 343.929,Z 1145.406,A -85,B 0,C 180,E1 14979.216,E2 14979.216} C_VEL
LIN {X 0,Y 353.679,Z 1126.482,A -85,B 0,C 180,E1 14976.219,E2 14976.219} C_VEL
LIN {X 0,Y 363.852,Z 1105.79,A -85,B 0,C 180,E1 14973.485,E2 14973.485} C_VEL
LIN {X 0,Y 372.557,Z 1087.394,A -85,B 0,C 180,E1 14971.411,E2 14971.411} C_VEL
LIN {X 0,Y 381.736,Z 1067.04,A -85,B 0,C 180,E1 14969.435,E2 14969.435} C_VEL
LIN {X 0,Y 392.041,Z 1042.421,A -85,B 0,C 180,E1 14967.433,E2 14967.433} C_VEL
LIN {X 0,Y 400.366,Z 1020.773,A -85,B 0,C 180,E1 14965.965,E2 14965.965} C_VEL
LIN {X 0,Y 407.894,Z 999.575,A -85,B 0,C 180,E1 14964.741,E2 14964.741} C_VEL
LIN {X 0,Y 416.6,Z 972.484,A -85,B 0,C 180,E1 14963.446,E2 14963.446} C_VEL
LIN {X 0,Y 423.276,Z 948.736,A -85,B 0,C 180,E1 14962.537,E2 14962.537} C_VEL
LIN {X 0,Y 428.856,Z 926.233,A -85,B 0,C 180,E1 14961.832,E2 14961.832} C_VEL
LIN {X 0,Y 434.517,Z 899.009,A -85,B 0,C 180,E1 14961.125,E2 14961.125} C_VEL
LIN {X 0,Y 438.628,Z 870.939,A -85,B 0,C 180,E1 14960.524,E2 14960.524} C_VEL
LIN {X 0,Y 463.611,Z 638.054,A -85,B 0,C 180,E1 14956.437,E2 14956.437} C_VEL
LIN {X 0,Y 468.563,Z 593.048,A -85,B 0,C 180,E1 14955.661,E2 14955.661} C_VEL
LIN {X 0,Y 460.881,Z 580.152,A -85,B 0,C 180,E1 14952.944,E2 14952.944} C_VEL
LIN {X 0,Y 454.197,Z 569.107,A -85,B 0,C 180,E1 14950.336,E2 14950.336} C_VEL
LIN {X 0,Y 447.012,Z 557.832,A -85,B 0,C 180,E1 14947.261,E2 14947.261} C_VEL
LIN {X 0,Y 441.615,Z 549.516,A -85,B 0,C 180,E1 14944.675,E2 14944.675} C_VEL
LIN {X 0,Y 436.512,Z 541.67,A -85,B 0,C 180,E1 14941.969,E2 14941.969} C_VEL
LIN {X 0,Y 431.311,Z 534.015,A -85,B 0,C 180,E1 14938.937,E2 14938.937} C_VEL
LIN {X 0,Y 425.946,Z 526.142,A -85,B 0,C 180,E1 14935.355,E2 14935.355} C_VEL
LIN {X 0,Y 422.664,Z 521.409,A -85,B 0,C 180,E1 14932.865,E2 14932.865} C_VEL
LIN {X 0,Y 419.006,Z 516.051,A -85,B 0,C 180,E1 14929.69,E2 14929.69} C_VEL
LIN {X 0,Y 415.669,Z 510.912,A -85,B 0,C 180,E1 14926.223,E2 14926.223} C_VEL
LIN {X 0,Y 412.598,Z 506.573,A -85,B 0,C 180,E1 14922.512,E2 14922.512} C_VEL
LIN {X 0,Y 409.86,Z 504.388,A -85,B 0,C 180,E1 14918.734,E2 14918.734} C_VEL
LIN {X 0,Y 408.229,Z 501.616,A -85,B 0,C 180,E1 14915.325,E2 14915.325} C_VEL
LIN {X 0,Y 407.685,Z 500.541,A -85,B 0,C 180,E1 14913.645,E2 14913.645} C_VEL
LIN {X 0,Y 406.176,Z 499.772,A -85,B 0,C 180,E1 14909.2,E2 14909.2} C_VEL
LIN {X 0,Y 405.677,Z 499.448,A -85,B 0,C 180,E1 14905.16,E2 14905.16} C_VEL
LIN {X 0,Y 406.023,Z 499.621,A -85,B 0,C 180,E1 14900.37,E2 14900.37} C_VEL
LIN {X 0,Y 407.251,Z 500.244,A -85,B 0,C 180,E1 14895.986,E2 14895.986} C_VEL
LIN {X 0,Y 408.315,Z 501.058,A -85,B 0,C 180,E1 14893.543,E2 14893.543} C_VEL
LIN {X 0,Y 409.923,Z 504.086,A -85,B 0,C 180,E1 14890.228,E2 14890.228} C_VEL
LIN {X 0,Y 413.16,Z 506.71,A -85,B 0,C 180,E1 14886.021,E2 14886.021} C_VEL
LIN {X 0,Y 416.881,Z 511.746,A -85,B 0,C 180,E1 14882.01,E2 14882.01} C_VEL
LIN {X 0,Y 418.702,Z 513.378,A -85,B 0,C 180,E1 14880.415,E2 14880.415} C_VEL
LIN {X 0,Y 422.097,Z 517.81,A -85,B 0,C 180,E1 14877.63,E2 14877.63} C_VEL
LIN {X 0,Y 423.621,Z 519.455,A -85,B 0,C 180,E1 14876.546,E2 14876.546} C_VEL
LIN {X 0,Y 427.64,Z 524.222,A -85,B 0,C 180,E1 14873.86,E2 14873.86} C_VEL
LIN {X 0,Y 433.131,Z 531.299,A -85,B 0,C 180,E1 14870.612,E2 14870.612} C_VEL
LIN {X 0,Y 437.61,Z 536.965,A -85,B 0,C 180,E1 14868.276,E2 14868.276} C_VEL
LIN {X 0,Y 442.428,Z 543.223,A -85,B 0,C 180,E1 14866.005,E2 14866.005} C_VEL
LIN {X 0,Y 449.104,Z 552.164,A -85,B 0,C 180,E1 14863.126,E2 14863.126} C_VEL
LIN {X 0,Y 457.823,Z 564.102,A -85,B 0,C 180,E1 14859.808,E2 14859.808} C_VEL
LIN {X 0,Y 464.265,Z 573.702,A -85,B 0,C 180,E1 14857.567,E2 14857.567} C_VEL
LIN {X 0,Y 440.993,Z 790.108,A -85,B 0,C 180,E1 14853.829,E2 14853.829} C_VEL
LIN {X 0,Y 436.479,Z 820.61,A -85,B 0,C 180,E1 14853.106,E2 14853.106} C_VEL
LIN {X 0,Y 431.88,Z 844.747,A -85,B 0,C 180,E1 14852.366,E2 14852.366} C_VEL
LIN {X 0,Y 426.516,Z 868.55,A -85,B 0,C 180,E1 14851.478,E2 14851.478} C_VEL
LIN {X 0,Y 418.959,Z 896.768,A -85,B 0,C 180,E1 14850.187,E2 14850.187} C_VEL
LIN {X 0,Y 412.249,Z 918.502,A -85,B 0,C 180,E1 14848.988,E2 14848.988} C_VEL
LIN {X 0,Y 405.287,Z 938.797,A -85,B 0,C 180,E1 14847.692,E2 14847.692} C_VEL
LIN {X 0,Y 395.72,Z 963.947,A -85,B 0,C 180,E1 14845.798,E2 14845.798} C_VEL
LIN {X 0,Y 387.55,Z 983.302,A -85,B 0,C 180,E1 14844.077,E2 14844.077} C_VEL
LIN {X 0,Y 379.436,Z 1001.245,A -85,B 0,C 180,E1 14842.24,E2 14842.24} C_VEL
LIN {X 0,Y 371.234,Z 1018.322,A -85,B 0,C 180,E1 14840.231,E2 14840.231} C_VEL
LIN {X 0,Y 360.843,Z 1038.694,A -85,B 0,C 180,E1 14837.426,E2 14837.426} C_VEL
LIN {X 0,Y 351.702,Z 1055.488,A -85,B 0,C 180,E1 14834.669,E2 14834.669} C_VEL
LIN {X 0,Y 343.784,Z 1069.461,A -85,B 0,C 180,E1 14832.004,E2 14832.004} C_VEL
LIN {X 0,Y 335.556,Z 1083.678,A -85,B 0,C 180,E1 14828.857,E2 14828.857} C_VEL
LIN {X 0,Y 326.502,Z 1098.93,A -85,B 0,C 180,E1 14824.807,E2 14824.807} C_VEL
LIN {X 0,Y 320.201,Z 1109.528,A -85,B 0,C 180,E1 14821.461,E2 14821.461} C_VEL
LIN {X 0,Y 315.048,Z 1118.399,A -85,B 0,C 180,E1 14818.208,E2 14818.208} C_VEL
LIN {X 0,Y 310.319,Z 1126.825,A -85,B 0,C 180,E1 14814.608,E2 14814.608} C_VEL
LIN {X 0,Y 305.974,Z 1135.1,A -85,B 0,C 180,E1 14810.415,E2 14810.415} C_VEL
LIN {X 0,Y 302.195,Z 1143.071,A -85,B 0,C 180,E1 14805.348,E2 14805.348} C_VEL
LIN {X 0,Y 300.198,Z 1148.158,A -85,B 0,C 180,E1 14801.261,E2 14801.261} C_VEL
LIN {X 0,Y 298.989,Z 1151.92,A -85,B 0,C 180,E1 14797.492,E2 14797.492} C_VEL
LIN {X 0,Y 298.366,Z 1154.63,A -85,B 0,C 180,E1 14794.032,E2 14794.032} C_VEL
LIN {X 0,Y 298.286,Z 1155.166,A -85,B 0,C 180,E1 14793.217,E2 14793.217} C_VEL
LIN {X 0,Y 297.332,Z 1156.222,A -85,B 0,C 180,E1 14791.857,E2 14791.857} C_VEL
LIN {X 0,Y 293.179,Z 1158.087,A -85,B 0,C 180,E1 14789.402,E2 14789.402} C_VEL
LIN {X 0,Y 290.443,Z 1159.275,A -85,B 0,C 180,E1 14787.389,E2 14787.389} C_VEL
LIN {X 0,Y 290.128,Z 1159.544,A -85,B 0,C 180,E1 14786.51,E2 14786.51} C_VEL
LIN {X 0,Y 290.245,Z 1160.273,A -85,B 0,C 180,E1 14782.91,E2 14782.91} C_VEL
LIN {X 0,Y 290.669,Z 1160.338,A -85,B 0,C 180,E1 14778.92,E2 14778.92} C_VEL
LIN {X 0,Y 291.412,Z 1159.635,A -85,B 0,C 180,E1 14774.912,E2 14774.912} C_VEL
LIN {X 0,Y 292.71,Z 1158.128,A -85,B 0,C 180,E1 14770.829,E2 14770.829} C_VEL
LIN {X 0,Y 295.006,Z 1155.563,A -85,B 0,C 180,E1 14766.422,E2 14766.422} C_VEL
LIN {X 0,Y 299.382,Z 1150.956,A -85,B 0,C 180,E1 14760.957,E2 14760.957} C_VEL
LIN {X 0,Y 304.791,Z 1145.43,A -85,B 0,C 180,E1 14756.238,E2 14756.238} C_VEL
LIN {X 0,Y 311.432,Z 1139.016,A -85,B 0,C 180,E1 14751.879,E2 14751.879} C_VEL
LIN {X 0,Y 321.443,Z 1129.509,A -85,B 0,C 180,E1 14746.808,E2 14746.808} C_VEL
LIN {X 0,Y 332.836,Z 1119.014,A -85,B 0,C 180,E1 14742.337,E2 14742.337} C_VEL
LIN {X 0,Y 347.245,Z 1105.782,A -85,B 0,C 180,E1 14737.839,E2 14737.839} C_VEL
LIN {X 0,Y 365.789,Z 1089.429,A -85,B 0,C 180,E1 14733.365,E2 14733.365} C_VEL
LIN {X 0,Y 377.851,Z 1079.389,A -85,B 0,C 180,E1 14730.995,E2 14730.995} C_VEL
LIN {X 0,Y 359.705,Z 1102.263,A -85,B 0,C 180,E1 14727.675,E2 14727.675} C_VEL
LIN {X 0,Y 338.971,Z 1133.731,A -85,B 0,C 180,E1 14722.367,E2 14722.367} C_VEL
LIN {X 0,Y 326.492,Z 1155.105,A -85,B 0,C 180,E1 14718.089,E2 14718.089} C_VEL
LIN {X 0,Y 317.737,Z 1171.466,A -85,B 0,C 180,E1 14714.315,E2 14714.315} C_VEL
LIN {X 0,Y 309.606,Z 1187.74,A -85,B 0,C 180,E1 14709.991,E2 14709.991} C_VEL
LIN {X 0,Y 302.206,Z 1203.988,A -85,B 0,C 180,E1 14704.861,E2 14704.861} C_VEL
LIN {X 0,Y 297.74,Z 1215.151,A -85,B 0,C 180,E1 14700.694,E2 14700.694} C_VEL
LIN {X 0,Y 294.591,Z 1224.187,A -85,B 0,C 180,E1 14696.789,E2 14696.789} C_VEL
LIN {X 0,Y 292.311,Z 1232.242,A -85,B 0,C 180,E1 14692.738,E2 14692.738} C_VEL
LIN {X 0,Y 290.877,Z 1238.792,A -85,B 0,C 180,E1 14688.852,E2 14688.852} C_VEL
LIN {X 0,Y 290.166,Z 1243.942,A -85,B 0,C 180,E1 14685.182,E2 14685.182} C_VEL
LIN {X 0,Y 289.91,Z 1248.3,A -85,B 0,C 180,E1 14681.337,E2 14681.337} C_VEL
LIN {X 0,Y 289.941,Z 1251.507,A -85,B 0,C 180,E1 14677.53,E2 14677.53} C_VEL
LIN {X 0,Y 290.111,Z 1253.612,A -85,B 0,C 180,E1 14673.755,E2 14673.755} C_VEL
LIN {X 0,Y 290.138,Z 1254.561,A -85,B 0,C 180,E1 14670,E2 14670} C_VEL
LIN {X 0,Y 289.994,Z 1254.349,A -85,B 0,C 180,E1 14666.244,E2 14666.244} C_VEL
LIN {X 0,Y 289.731,Z 1252.988,A -85,B 0,C 180,E1 14662.464,E2 14662.464} C_VEL
LIN {X 0,Y 289.642,Z 1250.346,A -85,B 0,C 180,E1 14658.45,E2 14658.45} C_VEL
LIN {X 0,Y 289.983,Z 1246.222,A -85,B 0,C 180,E1 14654.16,E2 14654.16} C_VEL
LIN {X 0,Y 290.936,Z 1241.131,A -85,B 0,C 180,E1 14650.109,E2 14650.109} C_VEL
LIN {X 0,Y 292.72,Z 1234.768,A -85,B 0,C 180,E1 14646.016,E2 14646.016} C_VEL
LIN {X 0,Y 295.618,Z 1226.749,A -85,B 0,C 180,E1 14641.737,E2 14641.737} C_VEL
LIN {X 0,Y 300.784,Z 1214.756,A -85,B 0,C 180,E1 14636.508,E2 14636.508} C_VEL
LIN {X 0,Y 306.069,Z 1203.79,A -85,B 0,C 180,E1 14632.547,E2 14632.547} C_VEL
LIN {X 0,Y 312.05,Z 1192.159,A -85,B 0,C 180,E1 14628.939,E2 14628.939} C_VEL
LIN {X 0,Y 319.524,Z 1178.245,A -85,B 0,C 180,E1 14625.244,E2 14625.244} C_VEL
LIN {X 0,Y 328.992,Z 1160.676,A -85,B 0,C 180,E1 14621.35,E2 14621.35} C_VEL
LIN {X 0,Y 337.198,Z 1145.413,A -85,B 0,C 180,E1 14618.48,E2 14618.48} C_VEL
LIN {X 0,Y 345.892,Z 1129.039,A -85,B 0,C 180,E1 14615.821,E2 14615.821} C_VEL
LIN {X 0,Y 357.016,Z 1107.351,A -85,B 0,C 180,E1 14612.839,E2 14612.839} C_VEL
LIN {X 0,Y 366.504,Z 1087.808,A -85,B 0,C 180,E1 14610.601,E2 14610.601} C_VEL
LIN {X 0,Y 375.425,Z 1068.494,A -85,B 0,C 180,E1 14608.706,E2 14608.706} C_VEL
LIN {X 0,Y 385.69,Z 1044.873,A -85,B 0,C 180,E1 14606.736,E2 14606.736} C_VEL
LIN {X 0,Y 394.851,Z 1021.661,A -85,B 0,C 180,E1 14605.137,E2 14605.137} C_VEL
LIN {X 0,Y 402.507,Z 1000.683,A -85,B 0,C 180,E1 14603.914,E2 14603.914} C_VEL
LIN {X 0,Y 410.401,Z 977.074,A -85,B 0,C 180,E1 14602.757,E2 14602.757} C_VEL
LIN {X 0,Y 418.321,Z 950.039,A -85,B 0,C 180,E1 14601.69,E2 14601.69} C_VEL
LIN {X 0,Y 424.059,Z 927.58,A -85,B 0,C 180,E1 14600.978,E2 14600.978} C_VEL
LIN {X 0,Y 429.077,Z 904.504,A -85,B 0,C 180,E1 14600.371,E2 14600.371} C_VEL
LIN {X 0,Y 433.882,Z 875.508,A -85,B 0,C 180,E1 14599.715,E2 14599.715} C_VEL
LIN {X 0,Y 439.568,Z 824.129,A -85,B 0,C 180,E1 14598.78,E2 14598.78} C_VEL
LIN {X 0,Y 464.126,Z 603.256,A -85,B 0,C 180,E1 14594.95,E2 14594.95} C_VEL
LIN {X 0,Y 464.695,Z 597.736,A -85,B 0,C 180,E1 14594.836,E2 14594.836} C_VEL
LIN {X 0,Y 456.11,Z 583.108,A -85,B 0,C 180,E1 14591.668,E2 14591.668} C_VEL
LIN {X 0,Y 447.439,Z 569.143,A -85,B 0,C 180,E1 14588.093,E2 14588.093} C_VEL
LIN {X 0,Y 440.543,Z 558.374,A -85,B 0,C 180,E1 14584.881,E2 14584.881} C_VEL
LIN {X 0,Y 434.507,Z 549.168,A -85,B 0,C 180,E1 14581.714,E2 14581.714} C_VEL
LIN {X 0,Y 428.216,Z 539.718,A -85,B 0,C 180,E1 14577.968,E2 14577.968} C_VEL
LIN {X 0,Y 423.881,Z 533.486,A -85,B 0,C 180,E1 14574.993,E2 14574.993} C_VEL
LIN {X 0,Y 420.885,Z 529.027,A -85,B 0,C 180,E1 14572.629,E2 14572.629} C_VEL
LIN {X 0,Y 417.315,Z 523.759,A -85,B 0,C 180,E1 14569.508,E2 14569.508} C_VEL
LIN {X 0,Y 413.943,Z 518.61,A -85,B 0,C 180,E1 14566.022,E2 14566.022} C_VEL
LIN {X 0,Y 411.006,Z 514.399,A -85,B 0,C 180,E1 14562.442,E2 14562.442} C_VEL
LIN {X 0,Y 408.329,Z 512.283,A -85,B 0,C 180,E1 14558.751,E2 14558.751} C_VEL
LIN {X 0,Y 406.667,Z 509.494,A -85,B 0,C 180,E1 14555.292,E2 14555.292} C_VEL
LIN {X 0,Y 406.147,Z 508.402,A -85,B 0,C 180,E1 14553.652,E2 14553.652} C_VEL
LIN {X 0,Y 404.603,Z 507.615,A -85,B 0,C 180,E1 14549.067,E2 14549.067} C_VEL
LIN {X 0,Y 404.143,Z 507.293,A -85,B 0,C 180,E1 14544.971,E2 14544.971} C_VEL
LIN {X 0,Y 404.518,Z 507.493,A -85,B 0,C 180,E1 14540.193,E2 14540.193} C_VEL
LIN {X 0,Y 405.818,Z 508.125,A -85,B 0,C 180,E1 14535.79,E2 14535.79} C_VEL
LIN {X 0,Y 406.739,Z 508.831,A -85,B 0,C 180,E1 14533.692,E2 14533.692} C_VEL
LIN {X 0,Y 408.435,Z 512.004,A -85,B 0,C 180,E1 14530.199,E2 14530.199} C_VEL
LIN {X 0,Y 411.932,Z 514.953,A -85,B 0,C 180,E1 14525.716,E2 14525.716} C_VEL
LIN {X 0,Y 414.868,Z 519.178,A -85,B 0,C 180,E1 14522.483,E2 14522.483} C_VEL
LIN {X 0,Y 417.055,Z 521.188,A -85,B 0,C 180,E1 14520.548,E2 14520.548} C_VEL
LIN {X 0,Y 420.525,Z 525.646,A -85,B 0,C 180,E1 14517.707,E2 14517.707} C_VEL
LIN {X 0,Y 421.999,Z 527.338,A -85,B 0,C 180,E1 14516.647,E2 14516.647} C_VEL
LIN {X 0,Y 426.642,Z 532.998,A -85,B 0,C 180,E1 14513.552,E2 14513.552} C_VEL
LIN {X 0,Y 431.362,Z 539.058,A -85,B 0,C 180,E1 14510.772,E2 14510.772} C_VEL
LIN {X 0,Y 435.693,Z 544.54,A -85,B 0,C 180,E1 14508.507,E2 14508.507} C_VEL
LIN {X 0,Y 440.818,Z 551.258,A -85,B 0,C 180,E1 14506.065,E2 14506.065} C_VEL
LIN {X 0,Y 449.145,Z 562.41,A -85,B 0,C 180,E1 14502.536,E2 14502.536} C_VEL
LIN {X 0,Y 458.435,Z 575.64,A -85,B 0,C 180,E1 14499.067,E2 14499.067} C_VEL
LIN {X 0,Y 460.359,Z 578.808,A -85,B 0,C 180,E1 14498.385,E2 14498.385} C_VEL
LIN {X 0,Y 436.745,Z 792.303,A -85,B 0,C 180,E1 14494.695,E2 14494.695} C_VEL
LIN {X 0,Y 432.102,Z 822.537,A -85,B 0,C 180,E1 14493.969,E2 14493.969} C_VEL
LIN {X 0,Y 427.414,Z 846.515,A -85,B 0,C 180,E1 14493.229,E2 14493.229} C_VEL
LIN {X 0,Y 421.275,Z 872.983,A -85,B 0,C 180,E1 14492.23,E2 14492.23} C_VEL
LIN {X 0,Y 414.022,Z 898.937,A -85,B 0,C 180,E1 14491.018,E2 14491.018} C_VEL
LIN {X 0,Y 407.424,Z 919.898,A -85,B 0,C 180,E1 14489.859,E2 14489.859} C_VEL
LIN {X 0,Y 400.093,Z 940.884,A -85,B 0,C 180,E1 14488.516,E2 14488.516} C_VEL
LIN {X 0,Y 389.973,Z 966.788,A -85,B 0,C 180,E1 14486.546,E2 14486.546} C_VEL
LIN {X 0,Y 382.016,Z 985.188,A -85,B 0,C 180,E1 14484.895,E2 14484.895} C_VEL
LIN {X 0,Y 373.711,Z 1003.1,A -85,B 0,C 180,E1 14483.046,E2 14483.046} C_VEL
LIN {X 0,Y 363.811,Z 1023.2,A -85,B 0,C 180,E1 14480.636,E2 14480.636} C_VEL
LIN {X 0,Y 353.539,Z 1042.421,A -85,B 0,C 180,E1 14477.875,E2 14477.875} C_VEL
LIN {X 0,Y 345.162,Z 1057.394,A -85,B 0,C 180,E1 14475.366,E2 14475.366} C_VEL
LIN {X 0,Y 337.195,Z 1071.128,A -85,B 0,C 180,E1 14472.715,E2 14472.715} C_VEL
LIN {X 0,Y 328.004,Z 1086.684,A -85,B 0,C 180,E1 14469.208,E2 14469.208} C_VEL
LIN {X 0,Y 319.413,Z 1100.583,A -85,B 0,C 180,E1 14465.397,E2 14465.397} C_VEL
LIN {X 0,Y 313.228,Z 1110.656,A -85,B 0,C 180,E1 14462.159,E2 14462.159} C_VEL
LIN {X 0,Y 307.693,Z 1119.85,A -85,B 0,C 180,E1 14458.722,E2 14458.722} C_VEL
LIN {X 0,Y 302.969,Z 1127.963,A -85,B 0,C 180,E1 14455.184,E2 14455.184} C_VEL
LIN {X 0,Y 298.748,Z 1135.638,A -85,B 0,C 180,E1 14451.246,E2 14451.246} C_VEL
LIN {X 0,Y 294.676,Z 1143.922,A -85,B 0,C 180,E1 14446.002,E2 14446.002} C_VEL
LIN {X 0,Y 292.416,Z 1149.379,A -85,B 0,C 180,E1 14441.557,E2 14441.557} C_VEL
LIN {X 0,Y 291.084,Z 1153.381,A -85,B 0,C 180,E1 14437.446,E2 14437.446} C_VEL
LIN {X 0,Y 290.454,Z 1156.067,A -85,B 0,C 180,E1 14433.896,E2 14433.896} C_VEL
LIN {X 0,Y 290.195,Z 1158.173,A -85,B 0,C 180,E1 14430.137,E2 14430.137} C_VEL
LIN {X 0,Y 290.128,Z 1159.544,A -85,B 0,C 180,E1 14426.51,E2 14426.51} C_VEL
LIN {X 0,Y 289.347,Z 1160.078,A -85,B 0,C 180,E1 14425.098,E2 14425.098} C_VEL
LIN {X 0,Y 285.676,Z 1161.212,A -85,B 0,C 180,E1 14422.648,E2 14422.648} C_VEL
LIN {X 0,Y 282.973,Z 1161.86,A -85,B 0,C 180,E1 14420.453,E2 14420.453} C_VEL
LIN {X 0,Y 282.724,Z 1161.862,A -85,B 0,C 180,E1 14419.547,E2 14419.547} C_VEL
LIN {X 0,Y 283.556,Z 1161.23,A -85,B 0,C 180,E1 14414.917,E2 14414.917} C_VEL
LIN {X 0,Y 285.006,Z 1159.762,A -85,B 0,C 180,E1 14410.512,E2 14410.512} C_VEL
LIN {X 0,Y 287.19,Z 1157.563,A -85,B 0,C 180,E1 14406.397,E2 14406.397} C_VEL
LIN {X 0,Y 291.134,Z 1153.779,A -85,B 0,C 180,E1 14401.378,E2 14401.378} C_VEL
LIN {X 0,Y 297.305,Z 1147.995,A -85,B 0,C 180,E1 14395.95,E2 14395.95} C_VEL
LIN {X 0,Y 303.85,Z 1142.099,A -85,B 0,C 180,E1 14391.675,E2 14391.675} C_VEL
LIN {X 0,Y 313.653,Z 1133.612,A -85,B 0,C 180,E1 14386.731,E2 14386.731} C_VEL
LIN {X 0,Y 325.827,Z 1123.007,A -85,B 0,C 180,E1 14381.944,E2 14381.944} C_VEL
LIN {X 0,Y 341.743,Z 1109.588,A -85,B 0,C 180,E1 14377.099,E2 14377.099} C_VEL
LIN {X 0,Y 362.274,Z 1093.018,A -85,B 0,C 180,E1 14372.375,E2 14372.375} C_VEL
LIN {X 0,Y 368.756,Z 1088.182,A -85,B 0,C 180,E1 14371.141,E2 14371.141} C_VEL
LIN {X 0,Y 352.862,Z 1107.076,A -85,B 0,C 180,E1 14368.221,E2 14368.221} C_VEL
LIN {X 0,Y 331.977,Z 1136.462,A -85,B 0,C 180,E1 14362.953,E2 14362.953} C_VEL
LIN {X 0,Y 317.622,Z 1159.965,A -85,B 0,C 180,E1 14357.981,E2 14357.981} C_VEL
LIN {X 0,Y 306.835,Z 1179.117,A -85,B 0,C 180,E1 14353.117,E2 14353.117} C_VEL
LIN {X 0,Y 300.127,Z 1192.197,A -85,B 0,C 180,E1 14349.271,E2 14349.271} C_VEL
LIN {X 0,Y 294.736,Z 1203.552,A -85,B 0,C 180,E1 14345.458,E2 14345.458} C_VEL
LIN {X 0,Y 290.419,Z 1213.698,A -85,B 0,C 180,E1 14341.555,E2 14341.555} C_VEL
LIN {X 0,Y 287.091,Z 1222.643,A -85,B 0,C 180,E1 14337.594,E2 14337.594} C_VEL
LIN {X 0,Y 284.658,Z 1230.522,A -85,B 0,C 180,E1 14333.538,E2 14333.538} C_VEL
LIN {X 0,Y 283.127,Z 1237.027,A -85,B 0,C 180,E1 14329.603,E2 14329.603} C_VEL
LIN {X 0,Y 282.285,Z 1242.535,A -85,B 0,C 180,E1 14325.616,E2 14325.616} C_VEL
LIN {X 0,Y 281.994,Z 1246.892,A -85,B 0,C 180,E1 14321.66,E2 14321.66} C_VEL
LIN {X 0,Y 282.023,Z 1250.146,A -85,B 0,C 180,E1 14317.743,E2 14317.743} C_VEL
LIN {X 0,Y 282.21,Z 1252.178,A -85,B 0,C 180,E1 14314.063,E2 14314.063} C_VEL
LIN {X 0,Y 282.231,Z 1253.18,A -85,B 0,C 180,E1 14310.406,E2 14310.406} C_VEL
LIN {X 0,Y 282.119,Z 1253.09,A -85,B 0,C 180,E1 14306.546,E2 14306.546} C_VEL
LIN {X 0,Y 281.828,Z 1251.716,A -85,B 0,C 180,E1 14302.457,E2 14302.457} C_VEL
LIN {X 0,Y 281.726,Z 1249.101,A -85,B 0,C 180,E1 14298.328,E2 14298.328} C_VEL
LIN {X 0,Y 282.073,Z 1245.027,A -85,B 0,C 180,E1 14293.949,E2 14293.949} C_VEL
LIN {X 0,Y 283.012,Z 1240.191,A -85,B 0,C 180,E1 14289.959,E2 14289.959} C_VEL
LIN {X 0,Y 284.757,Z 1234.166,A -85,B 0,C 180,E1 14285.918,E2 14285.918} C_VEL
LIN {X 0,Y 287.506,Z 1226.745,A -85,B 0,C 180,E1 14281.772,E2 14281.772} C_VEL
LIN {X 0,Y 292.006,Z 1216.564,A -85,B 0,C 180,E1 14277.013,E2 14277.013} C_VEL
LIN {X 0,Y 298.066,Z 1204.308,A -85,B 0,C 180,E1 14272.344,E2 14272.344} C_VEL
LIN {X 0,Y 304.146,Z 1192.798,A -85,B 0,C 180,E1 14268.64,E2 14268.64} C_VEL
LIN {X 0,Y 310.935,Z 1180.496,A -85,B 0,C 180,E1 14265.232,E2 14265.232} C_VEL
LIN {X 0,Y 319.097,Z 1165.988,A -85,B 0,C 180,E1 14261.775,E2 14261.775} C_VEL
LIN {X 0,Y 329.756,Z 1146.842,A -85,B 0,C 180,E1 14257.967,E2 14257.967} C_VEL
LIN {X 0,Y 338.327,Z 1131.177,A -85,B 0,C 180,E1 14255.346,E2 14255.346} C_VEL
LIN {X 0,Y 347.243,Z 1114.415,A -85,B 0,C 180,E1 14252.927,E2 14252.927} C_VEL
LIN {X 0,Y 357.987,Z 1093.439,A -85,B 0,C 180,E1 14250.339,E2 14250.339} C_VEL
LIN {X 0,Y 368.407,Z 1071.558,A -85,B 0,C 180,E1 14248.107,E2 14248.107} C_VEL
LIN {X 0,Y 376.911,Z 1052.72,A -85,B 0,C 180,E1 14246.467,E2 14246.467} C_VEL
LIN {X 0,Y 385.784,Z 1031.669,A -85,B 0,C 180,E1 14244.888,E2 14244.888} C_VEL
LIN {X 0,Y 396.082,Z 1004.951,A -85,B 0,C 180,E1 14243.236,E2 14243.236} C_VEL
LIN {X 0,Y 403.744,Z 982.873,A -85,B 0,C 180,E1 14242.113,E2 14242.113} C_VEL
LIN {X 0,Y 410.917,Z 960.066,A -85,B 0,C 180,E1 14241.147,E2 14241.147} C_VEL
LIN {X 0,Y 418.993,Z 930.471,A -85,B 0,C 180,E1 14240.15,E2 14240.15} C_VEL
LIN {X 0,Y 424.463,Z 906.272,A -85,B 0,C 180,E1 14239.504,E2 14239.504} C_VEL
LIN {X 0,Y 428.986,Z 880.829,A -85,B 0,C 180,E1 14238.914,E2 14238.914} C_VEL
LIN {X 0,Y 433.757,Z 841.838,A -85,B 0,C 180,E1 14238.176,E2 14238.176} C_VEL
LIN {X 0,Y 458.587,Z 621.762,A -85,B 0,C 180,E1 14234.359,E2 14234.359} C_VEL
LIN {X 0,Y 460.83,Z 602.564,A -85,B 0,C 180,E1 14234.036,E2 14234.036} C_VEL
LIN {X 0,Y 452.307,Z 588.008,A -85,B 0,C 180,E1 14230.798,E2 14230.798} C_VEL
LIN {X 0,Y 444.09,Z 574.689,A -85,B 0,C 180,E1 14227.309,E2 14227.309} C_VEL
LIN {X 0,Y 437.705,Z 564.778,A -85,B 0,C 180,E1 14224.258,E2 14224.258} C_VEL
LIN {X 0,Y 432.499,Z 556.664,A -85,B 0,C 180,E1 14221.457,E2 14221.457} C_VEL
LIN {X 0,Y 427.145,Z 548.628,A -85,B 0,C 180,E1 14218.253,E2 14218.253} C_VEL
LIN {X 0,Y 422.238,Z 541.348,A -85,B 0,C 180,E1 14214.905,E2 14214.905} C_VEL
LIN {X 0,Y 418.959,Z 536.519,A -85,B 0,C 180,E1 14212.319,E2 14212.319} C_VEL
LIN {X 0,Y 415.599,Z 531.461,A -85,B 0,C 180,E1 14209.324,E2 14209.324} C_VEL
LIN {X 0,Y 412.201,Z 526.302,A -85,B 0,C 180,E1 14205.818,E2 14205.818} C_VEL
LIN {X 0,Y 409.343,Z 522.188,A -85,B 0,C 180,E1 14202.294,E2 14202.294} C_VEL
LIN {X 0,Y 406.754,Z 520.121,A -85,B 0,C 180,E1 14198.694,E2 14198.694} C_VEL
LIN {X 0,Y 405.108,Z 517.385,A -85,B 0,C 180,E1 14195.27,E2 14195.27} C_VEL
LIN {X 0,Y 404.641,Z 516.296,A -85,B 0,C 180,E1 14193.748,E2 14193.748} C_VEL
LIN {X 0,Y 403.076,Z 515.468,A -85,B 0,C 180,E1 14189.125,E2 14189.125} C_VEL
LIN {X 0,Y 402.604,Z 515.144,A -85,B 0,C 180,E1 14184.991,E2 14184.991} C_VEL
LIN {X 0,Y 402.987,Z 515.345,A -85,B 0,C 180,E1 14180.197,E2 14180.197} C_VEL
LIN {X 0,Y 404.305,Z 515.981,A -85,B 0,C 180,E1 14175.78,E2 14175.78} C_VEL
LIN {X 0,Y 405.209,Z 516.752,A -85,B 0,C 180,E1 14173.697,E2 14173.697} C_VEL
LIN {X 0,Y 407.008,Z 520.002,A -85,B 0,C 180,E1 14170.064,E2 14170.064} C_VEL
LIN {X 0,Y 410.292,Z 522.703,A -85,B 0,C 180,E1 14165.88,E2 14165.88} C_VEL
LIN {X 0,Y 413.219,Z 526.928,A -85,B 0,C 180,E1 14162.639,E2 14162.639} C_VEL
LIN {X 0,Y 415.343,Z 528.876,A -85,B 0,C 180,E1 14160.746,E2 14160.746} C_VEL
LIN {X 0,Y 418.796,Z 533.338,A -85,B 0,C 180,E1 14157.901,E2 14157.901} C_VEL
LIN {X 0,Y 420.286,Z 535.096,A -85,B 0,C 180,E1 14156.804,E2 14156.804} C_VEL
LIN {X 0,Y 424.874,Z 540.724,A -85,B 0,C 180,E1 14153.727,E2 14153.727} C_VEL
LIN {X 0,Y 429.481,Z 546.651,A -85,B 0,C 180,E1 14150.999,E2 14150.999} C_VEL
LIN {X 0,Y 433.965,Z 552.369,A -85,B 0,C 180,E1 14148.644,E2 14148.644} C_VEL
LIN {X 0,Y 440.145,Z 560.444,A -85,B 0,C 180,E1 14145.718,E2 14145.718} C_VEL
LIN {X 0,Y 448.512,Z 572.092,A -85,B 0,C 180,E1 14142.194,E2 14142.194} C_VEL
LIN {X 0,Y 456.266,Z 583.222,A -85,B 0,C 180,E1 14139.301,E2 14139.301} C_VEL
LIN {X 0,Y 456.461,Z 583.88,A -85,B 0,C 180,E1 14139.213,E2 14139.213} C_VEL
LIN {X 0,Y 432.808,Z 792.793,A -85,B 0,C 180,E1 14135.61,E2 14135.61} C_VEL
LIN {X 0,Y 428.047,Z 823.265,A -85,B 0,C 180,E1 14134.883,E2 14134.883} C_VEL
LIN {X 0,Y 423.273,Z 847.195,A -85,B 0,C 180,E1 14134.147,E2 14134.147} C_VEL
LIN {X 0,Y 417.264,Z 872.644,A -85,B 0,C 180,E1 14133.193,E2 14133.193} C_VEL
LIN {X 0,Y 409.711,Z 899.378,A -85,B 0,C 180,E1 14131.958,E2 14131.958} C_VEL
LIN {X 0,Y 402.755,Z 921.037,A -85,B 0,C 180,E1 14130.764,E2 14130.764} C_VEL
LIN {X 0,Y 395.265,Z 942.031,A -85,B 0,C 180,E1 14129.42,E2 14129.42} C_VEL
LIN {X 0,Y 385.033,Z 967.67,A -85,B 0,C 180,E1 14127.47,E2 14127.47} C_VEL
LIN {X 0,Y 376.53,Z 986.961,A -85,B 0,C 180,E1 14125.736,E2 14125.736} C_VEL
LIN {X 0,Y 367.822,Z 1005.365,A -85,B 0,C 180,E1 14123.825,E2 14123.825} C_VEL
LIN {X 0,Y 357.122,Z 1026.47,A -85,B 0,C 180,E1 14121.248,E2 14121.248} C_VEL
LIN {X 0,Y 347.252,Z 1044.407,A -85,B 0,C 180,E1 14118.625,E2 14118.625} C_VEL
LIN {X 0,Y 338.834,Z 1059.048,A -85,B 0,C 180,E1 14116.138,E2 14116.138} C_VEL
LIN {X 0,Y 330.008,Z 1073.851,A -85,B 0,C 180,E1 14113.227,E2 14113.227} C_VEL
LIN {X 0,Y 319.662,Z 1090.618,A -85,B 0,C 180,E1 14109.271,E2 14109.271} C_VEL
LIN {X 0,Y 312.144,Z 1102.511,A -85,B 0,C 180,E1 14105.916,E2 14105.916} C_VEL
LIN {X 0,Y 305.561,Z 1112.951,A -85,B 0,C 180,E1 14102.474,E2 14102.474} C_VEL
LIN {X 0,Y 299.416,Z 1122.924,A -85,B 0,C 180,E1 14098.604,E2 14098.604} C_VEL
LIN {X 0,Y 293.126,Z 1133.509,A -85,B 0,C 180,E1 14093.592,E2 14093.592} C_VEL
LIN {X 0,Y 289.23,Z 1140.597,A -85,B 0,C 180,E1 14089.465,E2 14089.465} C_VEL
LIN {X 0,Y 286.377,Z 1146.374,A -85,B 0,C 180,E1 14085.42,E2 14085.42} C_VEL
LIN {X 0,Y 284.493,Z 1150.935,A -85,B 0,C 180,E1 14081.53,E2 14081.53} C_VEL
LIN {X 0,Y 283.232,Z 1154.622,A -85,B 0,C 180,E1 14077.643,E2 14077.643} C_VEL
LIN {X 0,Y 282.57,Z 1157.343,A -85,B 0,C 180,E1 14073.993,E2 14073.993} C_VEL
LIN {X 0,Y 282.304,Z 1159.458,A -85,B 0,C 180,E1 14070.196,E2 14070.196} C_VEL
LIN {X 0,Y 282.251,Z 1160.929,A -85,B 0,C 180,E1 14066.284,E2 14066.284} C_VEL
LIN {X 0,Y 282.391,Z 1161.687,A -85,B 0,C 180,E1 14062.462,E2 14062.462} C_VEL
LIN {X 0,Y 282.724,Z 1161.862,A -85,B 0,C 180,E1 14059.547,E2 14059.547} C_VEL
LIN {X 0,Y 281.969,Z 1161.932,A -85,B 0,C 180,E1 14057.981,E2 14057.981} C_VEL
LIN {X 0,Y 276.621,Z 1162.403,A -85,B 0,C 180,E1 14053.513,E2 14053.513} C_VEL
LIN {X 0,Y 276.452,Z 1162.231,A -85,B 0,C 180,E1 14052.357,E2 14052.357} C_VEL
LIN {X 0,Y 279.247,Z 1159.703,A -85,B 0,C 180,E1 14046.58,E2 14046.58} C_VEL
LIN {X 0,Y 282.863,Z 1156.468,A -85,B 0,C 180,E1 14041.823,E2 14041.823} C_VEL
LIN {X 0,Y 288.045,Z 1152.059,A -85,B 0,C 180,E1 14037.015,E2 14037.015} C_VEL
LIN {X 0,Y 296.602,Z 1144.939,A -85,B 0,C 180,E1 14031.274,E2 14031.274} C_VEL
LIN {X 0,Y 306.728,Z 1136.78,A -85,B 0,C 180,E1 14026.233,E2 14026.233} C_VEL
LIN {X 0,Y 320.376,Z 1125.859,A -85,B 0,C 180,E1 14021.022,E2 14021.022} C_VEL
LIN {X 0,Y 336.346,Z 1113.484,A -85,B 0,C 180,E1 14016.339,E2 14016.339} C_VEL
LIN {X 0,Y 357.003,Z 1098.217,A -85,B 0,C 180,E1 14011.749,E2 14011.749} C_VEL
LIN {X 0,Y 359.316,Z 1096.585,A -85,B 0,C 180,E1 14011.271,E2 14011.271} C_VEL
LIN {X 0,Y 340.198,Z 1118.802,A -85,B 0,C 180,E1 14007.514,E2 14007.514} C_VEL
LIN {X 0,Y 318.822,Z 1148.413,A -85,B 0,C 180,E1 14001.613,E2 14001.613} C_VEL
LIN {X 0,Y 306.031,Z 1168.76,A -85,B 0,C 180,E1 13996.768,E2 13996.768} C_VEL
LIN {X 0,Y 295.155,Z 1187.808,A -85,B 0,C 180,E1 13991.345,E2 13991.345} C_VEL
LIN {X 0,Y 288.344,Z 1201.071,A -85,B 0,C 180,E1 13986.863,E2 13986.863} C_VEL
LIN {X 0,Y 283.375,Z 1211.78,A -85,B 0,C 180,E1 13982.673,E2 13982.673} C_VEL
LIN {X 0,Y 279.769,Z 1220.77,A -85,B 0,C 180,E1 13978.614,E2 13978.614} C_VEL
LIN {X 0,Y 277.116,Z 1228.602,A -85,B 0,C 180,E1 13974.515,E2 13974.515} C_VEL
LIN {X 0,Y 275.376,Z 1235.289,A -85,B 0,C 180,E1 13970.4,E2 13970.4} C_VEL
LIN {X 0,Y 274.426,Z 1240.849,A -85,B 0,C 180,E1 13966.293,E2 13966.293} C_VEL
LIN {X 0,Y 274.064,Z 1245.418,A -85,B 0,C 180,E1 13962.104,E2 13962.104} C_VEL
LIN {X 0,Y 274.091,Z 1248.625,A -85,B 0,C 180,E1 13958.179,E2 13958.179} C_VEL
LIN {X 0,Y 274.305,Z 1250.753,A -85,B 0,C 180,E1 13954.39,E2 13954.39} C_VEL
LIN {X 0,Y 274.34,Z 1251.818,A -85,B 0,C 180,E1 13950.626,E2 13950.626} C_VEL
LIN {X 0,Y 274.236,Z 1251.772,A -85,B 0,C 180,E1 13946.656,E2 13946.656} C_VEL
LIN {X 0,Y 273.939,Z 1250.549,A -85,B 0,C 180,E1 13942.66,E2 13942.66} C_VEL
LIN {X 0,Y 273.81,Z 1247.802,A -85,B 0,C 180,E1 13938.147,E2 13938.147} C_VEL
LIN {X 0,Y 274.137,Z 1244.022,A -85,B 0,C 180,E1 13933.907,E2 13933.907} C_VEL
LIN {X 0,Y 275.158,Z 1238.969,A -85,B 0,C 180,E1 13929.583,E2 13929.583} C_VEL
LIN {X 0,Y 276.978,Z 1233.019,A -85,B 0,C 180,E1 13925.467,E2 13925.467} C_VEL
LIN {X 0,Y 279.906,Z 1225.516,A -85,B 0,C 180,E1 13921.168,E2 13921.168} C_VEL
LIN {X 0,Y 284.638,Z 1215.3,A -85,B 0,C 180,E1 13916.288,E2 13916.288} C_VEL
LIN {X 0,Y 290.937,Z 1203.068,A -85,B 0,C 180,E1 13911.534,E2 13911.534} C_VEL
LIN {X 0,Y 297.403,Z 1191.367,A -85,B 0,C 180,E1 13907.702,E2 13907.702} C_VEL
LIN {X 0,Y 304.41,Z 1179.16,A -85,B 0,C 180,E1 13904.271,E2 13904.271} C_VEL
LIN {X 0,Y 313.355,Z 1163.812,A -85,B 0,C 180,E1 13900.586,E2 13900.586} C_VEL
LIN {X 0,Y 323.91,Z 1145.32,A -85,B 0,C 180,E1 13896.917,E2 13896.917} C_VEL
LIN {X 0,Y 332.931,Z 1129.28,A -85,B 0,C 180,E1 13894.23,E2 13894.23} C_VEL
LIN {X 0,Y 342.541,Z 1111.675,A -85,B 0,C 180,E1 13891.697,E2 13891.697} C_VEL
LIN {X 0,Y 354.708,Z 1088.18,A -85,B 0,C 180,E1 13888.878,E2 13888.878} C_VEL
LIN {X 0,Y 364.148,Z 1068.805,A -85,B 0,C 180,E1 13886.94,E2 13886.94} C_VEL
LIN {X 0,Y 373.594,Z 1048.234,A -85,B 0,C 180,E1 13885.186,E2 13885.186} C_VEL
LIN {X 0,Y 384.865,Z 1021.312,A -85,B 0,C 180,E1 13883.285,E2 13883.285} C_VEL
LIN {X 0,Y 393.026,Z 999.871,A -85,B 0,C 180,E1 13882.038,E2 13882.038} C_VEL
LIN {X 0,Y 401.036,Z 976.85,A -85,B 0,C 180,E1 13880.917,E2 13880.917} C_VEL
LIN {X 0,Y 409.653,Z 948.725,A -85,B 0,C 180,E1 13879.813,E2 13879.813} C_VEL
LIN {X 0,Y 416.003,Z 924.679,A -85,B 0,C 180,E1 13879.069,E2 13879.069} C_VEL
LIN {X 0,Y 421.382,Z 900.408,A -85,B 0,C 180,E1 13878.441,E2 13878.441} C_VEL
LIN {X 0,Y 426.346,Z 870.23,A -85,B 0,C 180,E1 13877.779,E2 13877.779} C_VEL
LIN {X 0,Y 445.288,Z 705.48,A -85,B 0,C 180,E1 13874.874,E2 13874.874} C_VEL
LIN {X 0,Y 456.908,Z 607.285,A -85,B 0,C 180,E1 13873.188,E2 13873.188} C_VEL
LIN {X 0,Y 449.079,Z 593.889,A -85,B 0,C 180,E1 13870.131,E2 13870.131} C_VEL
LIN {X 0,Y 441.633,Z 581.645,A -85,B 0,C 180,E1 13866.892,E2 13866.892} C_VEL
LIN {X 0,Y 435.694,Z 572.309,A -85,B 0,C 180,E1 13864.014,E2 13864.014} C_VEL
LIN {X 0,Y 430.5,Z 564.16,A -85,B 0,C 180,E1 13861.198,E2 13861.198} C_VEL
LIN {X 0,Y 425.726,Z 556.941,A -85,B 0,C 180,E1 13858.318,E2 13858.318} C_VEL
LIN {X 0,Y 420.393,Z 548.951,A -85,B 0,C 180,E1 13854.678,E2 13854.678} C_VEL
LIN {X 0,Y 417.304,Z 544.335,A -85,B 0,C 180,E1 13852.219,E2 13852.219} C_VEL
LIN {X 0,Y 413.848,Z 539.152,A -85,B 0,C 180,E1 13849.137,E2 13849.137} C_VEL
LIN {X 0,Y 410.464,Z 533.995,A -85,B 0,C 180,E1 13845.613,E2 13845.613} C_VEL
LIN {X 0,Y 407.656,Z 529.961,A -85,B 0,C 180,E1 13842.113,E2 13842.113} C_VEL
LIN {X 0,Y 405.237,Z 528.034,A -85,B 0,C 180,E1 13838.733,E2 13838.733} C_VEL
LIN {X 0,Y 403.548,Z 525.275,A -85,B 0,C 180,E1 13835.245,E2 13835.245} C_VEL
LIN {X 0,Y 403.031,Z 524.09,A -85,B 0,C 180,E1 13833.586,E2 13833.586} C_VEL
LIN {X 0,Y 401.538,Z 523.319,A -85,B 0,C 180,E1 13829.138,E2 13829.138} C_VEL
LIN {X 0,Y 401.065,Z 522.996,A -85,B 0,C 180,E1 13825.011,E2 13825.011} C_VEL
LIN {X 0,Y 401.473,Z 523.209,A -85,B 0,C 180,E1 13820.092,E2 13820.092} C_VEL
LIN {X 0,Y 402.877,Z 523.864,A -85,B 0,C 180,E1 13815.582,E2 13815.582} C_VEL
LIN {X 0,Y 403.673,Z 524.671,A -85,B 0,C 180,E1 13813.715,E2 13813.715} C_VEL
LIN {X 0,Y 405.631,Z 528.047,A -85,B 0,C 180,E1 13809.859,E2 13809.859} C_VEL
LIN {X 0,Y 408.742,Z 530.635,A -85,B 0,C 180,E1 13805.932,E2 13805.932} C_VEL
LIN {X 0,Y 411.796,Z 534.891,A -85,B 0,C 180,E1 13802.588,E2 13802.588} C_VEL
LIN {X 0,Y 413.682,Z 536.647,A -85,B 0,C 180,E1 13800.901,E2 13800.901} C_VEL
LIN {X 0,Y 417.175,Z 541.126,A -85,B 0,C 180,E1 13798.019,E2 13798.019} C_VEL
LIN {X 0,Y 418.761,Z 543.13,A -85,B 0,C 180,E1 13796.826,E2 13796.826} C_VEL
LIN {X 0,Y 423.069,Z 548.385,A -85,B 0,C 180,E1 13793.931,E2 13793.931} C_VEL
LIN {X 0,Y 427.566,Z 554.185,A -85,B 0,C 180,E1 13791.252,E2 13791.252} C_VEL
LIN {X 0,Y 432.121,Z 560.029,A -85,B 0,C 180,E1 13788.845,E2 13788.845} C_VEL
LIN {X 0,Y 438.178,Z 568.09,A -85,B 0,C 180,E1 13785.93,E2 13785.93} C_VEL
LIN {X 0,Y 446.002,Z 579.043,A -85,B 0,C 180,E1 13782.596,E2 13782.596} C_VEL
LIN {X 0,Y 452.642,Z 588.637,A -85,B 0,C 180,E1 13780.058,E2 13780.058} C_VEL
LIN {X 0,Y 428.959,Z 793.002,A -85,B 0,C 180,E1 13776.543,E2 13776.543} C_VEL
LIN {X 0,Y 424.108,Z 823.653,A -85,B 0,C 180,E1 13775.818,E2 13775.818} C_VEL
LIN {X 0,Y 419.228,Z 847.76,A -85,B 0,C 180,E1 13775.083,E2 13775.083} C_VEL
LIN {X 0,Y 413.293,Z 872.557,A -85,B 0,C 180,E1 13774.162,E2 13774.162} C_VEL
LIN {X 0,Y 405.482,Z 899.909,A -85,B 0,C 180,E1 13772.913,E2 13772.913} C_VEL
LIN {X 0,Y 398.404,Z 921.556,A -85,B 0,C 180,E1 13771.726,E2 13771.726} C_VEL
LIN {X 0,Y 390.97,Z 942.012,A -85,B 0,C 180,E1 13770.426,E2 13770.426} C_VEL
LIN {X 0,Y 380.595,Z 967.646,A -85,B 0,C 180,E1 13768.495,E2 13768.495} C_VEL
LIN {X 0,Y 371.885,Z 987.041,A -85,B 0,C 180,E1 13766.763,E2 13766.763} C_VEL
LIN {X 0,Y 363.376,Z 1004.699,A -85,B 0,C 180,E1 13764.944,E2 13764.944} C_VEL
LIN {X 0,Y 353.69,Z 1023.568,A -85,B 0,C 180,E1 13762.691,E2 13762.691} C_VEL
LIN {X 0,Y 342.393,Z 1043.952,A -85,B 0,C 180,E1 13759.784,E2 13759.784} C_VEL
LIN {X 0,Y 333.296,Z 1059.473,A -85,B 0,C 180,E1 13757.164,E2 13757.164} C_VEL
LIN {X 0,Y 324.849,Z 1073.287,A -85,B 0,C 180,E1 13754.456,E2 13754.456} C_VEL
LIN {X 0,Y 315.045,Z 1088.931,A -85,B 0,C 180,E1 13750.855,E2 13750.855} C_VEL
LIN {X 0,Y 306.182,Z 1102.467,A -85,B 0,C 180,E1 13747.062,E2 13747.062} C_VEL
LIN {X 0,Y 299.256,Z 1113.065,A -85,B 0,C 180,E1 13743.568,E2 13743.568} C_VEL
LIN {X 0,Y 293.597,Z 1121.866,A -85,B 0,C 180,E1 13740.184,E2 13740.184} C_VEL
LIN {X 0,Y 288.543,Z 1129.942,A -85,B 0,C 180,E1 13736.566,E2 13736.566} C_VEL
LIN {X 0,Y 283.884,Z 1137.782,A -85,B 0,C 180,E1 13732.419,E2 13732.419} C_VEL
LIN {X 0,Y 279.554,Z 1145.902,A -85,B 0,C 180,E1 13727.158,E2 13727.158} C_VEL
LIN {X 0,Y 276.868,Z 1151.793,A -85,B 0,C 180,E1 13722.201,E2 13722.201} C_VEL
LIN {X 0,Y 275.386,Z 1155.881,A -85,B 0,C 180,E1 13717.852,E2 13717.852} C_VEL
LIN {X 0,Y 274.667,Z 1158.754,A -85,B 0,C 180,E1 13713.902,E2 13713.902} C_VEL
LIN {X 0,Y 274.397,Z 1160.882,A -85,B 0,C 180,E1 13709.949,E2 13709.949} C_VEL
LIN {X 0,Y 274.377,Z 1162.362,A -85,B 0,C 180,E1 13705.828,E2 13705.828} C_VEL
LIN {X 0,Y 274.551,Z 1163.09,A -85,B 0,C 180,E1 13702.032,E2 13702.032} C_VEL
LIN {X 0,Y 275.024,Z 1163.206,A -85,B 0,C 180,E1 13698.22,E2 13698.22} C_VEL
LIN {X 0,Y 275.932,Z 1162.616,A -85,B 0,C 180,E1 13694.051,E2 13694.051} C_VEL
LIN {X 0,Y 276.452,Z 1162.231,A -85,B 0,C 180,E1 13692.357,E2 13692.357} C_VEL
LIN {X 0,Y 276.081,Z 1162.005,A -85,B 0,C 180,E1 13690.749,E2 13690.749} C_VEL
LIN {X 0,Y 272.223,Z 1161.4,A -85,B 0,C 180,E1 13686.257,E2 13686.257} C_VEL
LIN {X 0,Y 272.438,Z 1160.819,A -85,B 0,C 180,E1 13684.974,E2 13684.974} C_VEL
LIN {X 0,Y 276.551,Z 1157.593,A -85,B 0,C 180,E1 13680.207,E2 13680.207} C_VEL
LIN {X 0,Y 284.047,Z 1151.807,A -85,B 0,C 180,E1 13674.141,E2 13674.141} C_VEL
LIN {X 0,Y 292.129,Z 1145.678,A -85,B 0,C 180,E1 13669.349,E2 13669.349} C_VEL
LIN {X 0,Y 303.64,Z 1137.192,A -85,B 0,C 180,E1 13664.138,E2 13664.138} C_VEL
LIN {X 0,Y 320.353,Z 1125.098,A -85,B 0,C 180,E1 13658.451,E2 13658.451} C_VEL
LIN {X 0,Y 341.967,Z 1109.99,A -85,B 0,C 180,E1 13653.05,E2 13653.05} C_VEL
LIN {X 0,Y 349.92,Z 1104.655,A -85,B 0,C 180,E1 13651.396,E2 13651.396} C_VEL
LIN {X 0,Y 330.715,Z 1125.99,A -85,B 0,C 180,E1 13647.514,E2 13647.514} C_VEL
LIN {X 0,Y 308.4,Z 1155.7,A -85,B 0,C 180,E1 13641.088,E2 13641.088} C_VEL
LIN {X 0,Y 296.143,Z 1174.316,A -85,B 0,C 180,E1 13636.199,E2 13636.199} C_VEL
LIN {X 0,Y 287.832,Z 1188.18,A -85,B 0,C 180,E1 13631.977,E2 13631.977} C_VEL
LIN {X 0,Y 281.186,Z 1200.333,A -85,B 0,C 180,E1 13627.706,E2 13627.706} C_VEL
LIN {X 0,Y 275.974,Z 1210.908,A -85,B 0,C 180,E1 13623.415,E2 13623.415} C_VEL
LIN {X 0,Y 271.984,Z 1220.235,A -85,B 0,C 180,E1 13619.03,E2 13619.03} C_VEL
LIN {X 0,Y 269.12,Z 1228.312,A -85,B 0,C 180,E1 13614.59,E2 13614.59} C_VEL
LIN {X 0,Y 267.373,Z 1234.831,A -85,B 0,C 180,E1 13610.352,E2 13610.352} C_VEL
LIN {X 0,Y 266.415,Z 1240.495,A -85,B 0,C 180,E1 13605.901,E2 13605.901} C_VEL
LIN {X 0,Y 266.131,Z 1244.904,A -85,B 0,C 180,E1 13601.486,E2 13601.486} C_VEL
LIN {X 0,Y 266.213,Z 1247.819,A -85,B 0,C 180,E1 13597.554,E2 13597.554} C_VEL
LIN {X 0,Y 266.424,Z 1249.536,A -85,B 0,C 180,E1 13594.089,E2 13594.089} C_VEL
LIN {X 0,Y 266.463,Z 1250.464,A -85,B 0,C 180,E1 13590.43,E2 13590.43} C_VEL
LIN {X 0,Y 266.344,Z 1250.403,A -85,B 0,C 180,E1 13586.556,E2 13586.556} C_VEL
LIN {X 0,Y 266.026,Z 1249.155,A -85,B 0,C 180,E1 13582.441,E2 13582.441} C_VEL
LIN {X 0,Y 265.892,Z 1246.452,A -85,B 0,C 180,E1 13577.888,E2 13577.888} C_VEL
LIN {X 0,Y 266.267,Z 1242.543,A -85,B 0,C 180,E1 13573.418,E2 13573.418} C_VEL
LIN {X 0,Y 267.314,Z 1237.715,A -85,B 0,C 180,E1 13569.185,E2 13569.185} C_VEL
LIN {X 0,Y 269.239,Z 1231.755,A -85,B 0,C 180,E1 13564.953,E2 13564.953} C_VEL
LIN {X 0,Y 272.154,Z 1224.643,A -85,B 0,C 180,E1 13560.749,E2 13560.749} C_VEL
LIN {X 0,Y 276.42,Z 1215.696,A -85,B 0,C 180,E1 13556.303,E2 13556.303} C_VEL
LIN {X 0,Y 283.274,Z 1202.932,A -85,B 0,C 180,E1 13551.076,E2 13551.076} C_VEL
LIN {X 0,Y 290.228,Z 1190.786,A -85,B 0,C 180,E1 13546.989,E2 13546.989} C_VEL
LIN {X 0,Y 297.534,Z 1178.465,A -85,B 0,C 180,E1 13543.458,E2 13543.458} C_VEL
LIN {X 0,Y 306.275,Z 1163.923,A -85,B 0,C 180,E1 13539.898,E2 13539.898} C_VEL
LIN {X 0,Y 317.634,Z 1144.721,A -85,B 0,C 180,E1 13536.001,E2 13536.001} C_VEL
LIN {X 0,Y 327.089,Z 1128.401,A -85,B 0,C 180,E1 13533.237,E2 13533.237} C_VEL
LIN {X 0,Y 336.965,Z 1110.807,A -85,B 0,C 180,E1 13530.689,E2 13530.689} C_VEL
LIN {X 0,Y 349.467,Z 1087.229,A -85,B 0,C 180,E1 13527.86,E2 13527.86} C_VEL
LIN {X 0,Y 359.131,Z 1067.776,A -85,B 0,C 180,E1 13525.92,E2 13525.92} C_VEL
LIN {X 0,Y 368.79,Z 1047.127,A -85,B 0,C 180,E1 13524.167,E2 13524.167} C_VEL
LIN {X 0,Y 380.035,Z 1020.867,A -85,B 0,C 180,E1 13522.319,E2 13522.319} C_VEL
LIN {X 0,Y 388.42,Z 999.294,A -85,B 0,C 180,E1 13521.068,E2 13521.068} C_VEL
LIN {X 0,Y 395.927,Z 978.217,A -85,B 0,C 180,E1 13520.041,E2 13520.041} C_VEL
LIN {X 0,Y 404.423,Z 951.629,A -85,B 0,C 180,E1 13518.973,E2 13518.973} C_VEL
LIN {X 0,Y 411.45,Z 925.742,A -85,B 0,C 180,E1 13518.162,E2 13518.162} C_VEL
LIN {X 0,Y 416.698,Z 902.91,A -85,B 0,C 180,E1 13517.568,E2 13517.568} C_VEL
LIN {X 0,Y 421.752,Z 874.812,A -85,B 0,C 180,E1 13516.929,E2 13516.929} C_VEL
LIN {X 0,Y 427.53,Z 826.931,A -85,B 0,C 180,E1 13516.055,E2 13516.055} C_VEL
LIN {X 0,Y 453.18,Z 612.111,A -85,B 0,C 180,E1 13512.358,E2 13512.358} C_VEL
LIN {X 0,Y 445.699,Z 599.371,A -85,B 0,C 180,E1 13509.361,E2 13509.361} C_VEL
LIN {X 0,Y 438.8,Z 587.966,A -85,B 0,C 180,E1 13506.279,E2 13506.279} C_VEL
LIN {X 0,Y 433.181,Z 579.072,A -85,B 0,C 180,E1 13503.507,E2 13503.507} C_VEL
LIN {X 0,Y 428.633,Z 571.816,A -85,B 0,C 180,E1 13501.002,E2 13501.002} C_VEL
LIN {X 0,Y 423.971,Z 564.739,A -85,B 0,C 180,E1 13498.175,E2 13498.175} C_VEL
LIN {X 0,Y 418.795,Z 556.863,A -85,B 0,C 180,E1 13494.617,E2 13494.617} C_VEL
LIN {X 0,Y 415.458,Z 551.93,A -85,B 0,C 180,E1 13491.976,E2 13491.976} C_VEL
LIN {X 0,Y 412.1,Z 546.843,A -85,B 0,C 180,E1 13488.949,E2 13488.949} C_VEL
LIN {X 0,Y 408.879,Z 541.839,A -85,B 0,C 180,E1 13485.553,E2 13485.553} C_VEL
LIN {X 0,Y 406.097,Z 537.803,A -85,B 0,C 180,E1 13482.075,E2 13482.075} C_VEL
LIN {X 0,Y 403.647,Z 535.85,A -85,B 0,C 180,E1 13478.645,E2 13478.645} C_VEL
LIN {X 0,Y 401.962,Z 533.088,A -85,B 0,C 180,E1 13475.14,E2 13475.14} C_VEL
LIN {X 0,Y 401.458,Z 531.922,A -85,B 0,C 180,E1 13473.524,E2 13473.524} C_VEL
LIN {X 0,Y 399.973,Z 531.163,A -85,B 0,C 180,E1 13469.032,E2 13469.032} C_VEL
LIN {X 0,Y 399.532,Z 530.842,A -85,B 0,C 180,E1 13464.857,E2 13464.857} C_VEL
LIN {X 0,Y 399.954,Z 531.068,A -85,B 0,C 180,E1 13460.021,E2 13460.021} C_VEL
LIN {X 0,Y 401.364,Z 531.721,A -85,B 0,C 180,E1 13455.57,E2 13455.57} C_VEL
LIN {X 0,Y 402.1,Z 532.458,A -85,B 0,C 180,E1 13453.851,E2 13453.851} C_VEL
LIN {X 0,Y 404.088,Z 535.896,A -85,B 0,C 180,E1 13449.908,E2 13449.908} C_VEL
LIN {X 0,Y 407.101,Z 538.39,A -85,B 0,C 180,E1 13446.092,E2 13446.092} C_VEL
LIN {X 0,Y 410.134,Z 542.642,A -85,B 0,C 180,E1 13442.743,E2 13442.743} C_VEL
LIN {X 0,Y 412.024,Z 544.417,A -85,B 0,C 180,E1 13441.057,E2 13441.057} C_VEL
LIN {X 0,Y 415.784,Z 549.126,A -85,B 0,C 180,E1 13437.965,E2 13437.965} C_VEL
LIN {X 0,Y 421.273,Z 556.051,A -85,B 0,C 180,E1 13434.135,E2 13434.135} C_VEL
LIN {X 0,Y 425.69,Z 561.752,A -85,B 0,C 180,E1 13431.495,E2 13431.495} C_VEL
LIN {X 0,Y 430.363,Z 567.846,A -85,B 0,C 180,E1 13428.982,E2 13428.982} C_VEL
LIN {X 0,Y 436.185,Z 575.685,A -85,B 0,C 180,E1 13426.157,E2 13426.157} C_VEL
LIN {X 0,Y 443.599,Z 586.136,A -85,B 0,C 180,E1 13422.96,E2 13422.96} C_VEL
LIN {X 0,Y 448.86,Z 593.877,A -85,B 0,C 180,E1 13420.909,E2 13420.909} C_VEL
LIN {X 0,Y 424.921,Z 795.016,A -85,B 0,C 180,E1 13417.453,E2 13417.453} C_VEL
LIN {X 0,Y 419.961,Z 825.333,A -85,B 0,C 180,E1 13416.73,E2 13416.73} C_VEL
LIN {X 0,Y 414.934,Z 849.571,A -85,B 0,C 180,E1 13415.989,E2 13415.989} C_VEL
LIN {X 0,Y 408.296,Z 876.554,A -85,B 0,C 180,E1 13414.977,E2 13414.977} C_VEL
LIN {X 0,Y 400.552,Z 902.607,A -85,B 0,C 180,E1 13413.767,E2 13413.767} C_VEL
LIN {X 0,Y 393.072,Z 924.938,A -85,B 0,C 180,E1 13412.533,E2 13412.533} C_VEL
LIN {X 0,Y 383.66,Z 949.974,A -85,B 0,C 180,E1 13410.896,E2 13410.896} C_VEL
LIN {X 0,Y 374.651,Z 971.246,A -85,B 0,C 180,E1 13409.235,E2 13409.235} C_VEL
LIN {X 0,Y 366.285,Z 989.403,A -85,B 0,C 180,E1 13407.595,E2 13407.595} C_VEL
LIN {X 0,Y 356.999,Z 1008.161,A -85,B 0,C 180,E1 13405.635,E2 13405.635} C_VEL
LIN {X 0,Y 344.996,Z 1030.571,A -85,B 0,C 180,E1 13402.841,E2 13402.841} C_VEL
LIN {X 0,Y 335.636,Z 1046.827,A -85,B 0,C 180,E1 13400.431,E2 13400.431} C_VEL
LIN {X 0,Y 327.104,Z 1060.983,A -85,B 0,C 180,E1 13398.003,E2 13398.003} C_VEL
LIN {X 0,Y 318.44,Z 1074.805,A -85,B 0,C 180,E1 13395.265,E2 13395.265} C_VEL
LIN {X 0,Y 308.352,Z 1090.478,A -85,B 0,C 180,E1 13391.608,E2 13391.608} C_VEL
LIN {X 0,Y 299.243,Z 1104.03,A -85,B 0,C 180,E1 13387.755,E2 13387.755} C_VEL
LIN {X 0,Y 292.103,Z 1114.613,A -85,B 0,C 180,E1 13384.194,E2 13384.194} C_VEL
LIN {X 0,Y 285.809,Z 1124.09,A -85,B 0,C 180,E1 13380.444,E2 13380.444} C_VEL
LIN {X 0,Y 279.248,Z 1134.459,A -85,B 0,C 180,E1 13375.547,E2 13375.547} C_VEL
LIN {X 0,Y 274.244,Z 1142.715,A -85,B 0,C 180,E1 13370.62,E2 13370.62} C_VEL
LIN {X 0,Y 271.048,Z 1148.667,A -85,B 0,C 180,E1 13366.306,E2 13366.306} C_VEL
LIN {X 0,Y 268.985,Z 1153.23,A -85,B 0,C 180,E1 13362.286,E2 13362.286} C_VEL
LIN {X 0,Y 267.537,Z 1157.098,A -85,B 0,C 180,E1 13358.074,E2 13358.074} C_VEL
LIN {X 0,Y 266.806,Z 1159.893,A -85,B 0,C 180,E1 13354.205,E2 13354.205} C_VEL
LIN {X 0,Y 266.512,Z 1162.082,A -85,B 0,C 180,E1 13350.181,E2 13350.181} C_VEL
LIN {X 0,Y 266.48,Z 1163.633,A -85,B 0,C 180,E1 13346.041,E2 13346.041} C_VEL
LIN {X 0,Y 266.671,Z 1164.477,A -85,B 0,C 180,E1 13342.022,E2 13342.022} C_VEL
LIN {X 0,Y 267.212,Z 1164.654,A -85,B 0,C 180,E1 13337.869,E2 13337.869} C_VEL
LIN {X 0,Y 268.269,Z 1164.092,A -85,B 0,C 180,E1 13333.399,E2 13333.399} C_VEL
LIN {X 0,Y 270.155,Z 1162.65,A -85,B 0,C 180,E1 13328.728,E2 13328.728} C_VEL
LIN {X 0,Y 272.438,Z 1160.819,A -85,B 0,C 180,E1 13324.974,E2 13324.974} C_VEL
LIN {X 0,Y 272.685,Z 1160.193,A -85,B 0,C 180,E1 13323.347,E2 13323.347} C_VEL
LIN {X 0,Y 270.83,Z 1158.936,A -85,B 0,C 180,E1 13318.887,E2 13318.887} C_VEL
LIN {X 0,Y 271.657,Z 1157.955,A -85,B 0,C 180,E1 13317.506,E2 13317.506} C_VEL
LIN {X 0,Y 278.816,Z 1152.888,A -85,B 0,C 180,E1 13312.375,E2 13312.375} C_VEL
LIN {X 0,Y 288.891,Z 1146.058,A -85,B 0,C 180,E1 13306.999,E2 13306.999} C_VEL
LIN {X 0,Y 302.036,Z 1137.04,A -85,B 0,C 180,E1 13301.669,E2 13301.669} C_VEL
LIN {X 0,Y 319.378,Z 1125.598,A -85,B 0,C 180,E1 13296.376,E2 13296.376} C_VEL
LIN {X 0,Y 340.613,Z 1112.241,A -85,B 0,C 180,E1 13291.556,E2 13291.556} C_VEL
LIN {X 0,Y 320.576,Z 1133.689,A -85,B 0,C 180,E1 13287.344,E2 13287.344} C_VEL
LIN {X 0,Y 298.944,Z 1161.029,A -85,B 0,C 180,E1 13280.893,E2 13280.893} C_VEL
LIN {X 0,Y 284.611,Z 1182.175,A -85,B 0,C 180,E1 13274.792,E2 13274.792} C_VEL
LIN {X 0,Y 275.997,Z 1196.305,A -85,B 0,C 180,E1 13269.884,E2 13269.884} C_VEL
LIN {X 0,Y 269.988,Z 1207.31,A -85,B 0,C 180,E1 13265.436,E2 13265.436} C_VEL
LIN {X 0,Y 265.513,Z 1216.668,A -85,B 0,C 180,E1 13261.059,E2 13261.059} C_VEL
LIN {X 0,Y 262.293,Z 1224.638,A -85,B 0,C 180,E1 13256.732,E2 13256.732} C_VEL
LIN {X 0,Y 260.096,Z 1231.499,A -85,B 0,C 180,E1 13252.37,E2 13252.37} C_VEL
LIN {X 0,Y 258.745,Z 1237.528,A -85,B 0,C 180,E1 13247.775,E2 13247.775} C_VEL
LIN {X 0,Y 258.223,Z 1242.128,A -85,B 0,C 180,E1 13243.434,E2 13243.434} C_VEL
LIN {X 0,Y 258.219,Z 1245.595,A -85,B 0,C 180,E1 13239.135,E2 13239.135} C_VEL
LIN {X 0,Y 258.471,Z 1247.865,A -85,B 0,C 180,E1 13235.104,E2 13235.104} C_VEL
LIN {X 0,Y 258.577,Z 1249.056,A -85,B 0,C 180,E1 13231.108,E2 13231.108} C_VEL
LIN {X 0,Y 258.476,Z 1249.115,A -85,B 0,C 180,E1 13226.895,E2 13226.895} C_VEL
LIN {X 0,Y 258.137,Z 1247.921,A -85,B 0,C 180,E1 13222.576,E2 13222.576} C_VEL
LIN {X 0,Y 257.976,Z 1245.301,A -85,B 0,C 180,E1 13217.919,E2 13217.919} C_VEL
LIN {X 0,Y 258.338,Z 1241.495,A -85,B 0,C 180,E1 13213.357,E2 13213.357} C_VEL
LIN {X 0,Y 259.454,Z 1236.549,A -85,B 0,C 180,E1 13208.848,E2 13208.848} C_VEL
LIN {X 0,Y 261.477,Z 1230.611,A -85,B 0,C 180,E1 13204.485,E2 13204.485} C_VEL
LIN {X 0,Y 264.596,Z 1223.373,A -85,B 0,C 180,E1 13200.079,E2 13200.079} C_VEL
LIN {X 0,Y 269.005,Z 1214.574,A -85,B 0,C 180,E1 13195.599,E2 13195.599} C_VEL
LIN {X 0,Y 276.44,Z 1201.289,A -85,B 0,C 180,E1 13190.069,E2 13190.069} C_VEL
LIN {X 0,Y 283.58,Z 1189.353,A -85,B 0,C 180,E1 13185.997,E2 13185.997} C_VEL
LIN {X 0,Y 291.167,Z 1177.021,A -85,B 0,C 180,E1 13182.412,E2 13182.412} C_VEL
LIN {X 0,Y 300.739,Z 1161.651,A -85,B 0,C 180,E1 13178.619,E2 13178.619} C_VEL
LIN {X 0,Y 311.725,Z 1143.635,A -85,B 0,C 180,E1 13174.962,E2 13174.962} C_VEL
LIN {X 0,Y 321.39,Z 1127.369,A -85,B 0,C 180,E1 13172.197,E2 13172.197} C_VEL
LIN {X 0,Y 331.491,Z 1109.791,A -85,B 0,C 180,E1 13169.649,E2 13169.649} C_VEL
LIN {X 0,Y 344.369,Z 1086.097,A -85,B 0,C 180,E1 13166.804,E2 13166.804} C_VEL
LIN {X 0,Y 354.231,Z 1066.693,A -85,B 0,C 180,E1 13164.872,E2 13164.872} C_VEL
LIN {X 0,Y 364.183,Z 1045.864,A -85,B 0,C 180,E1 13163.11,E2 13163.11} C_VEL
LIN {X 0,Y 375.582,Z 1019.764,A -85,B 0,C 180,E1 13161.287,E2 13161.287} C_VEL
LIN {X 0,Y 384.21,Z 997.99,A -85,B 0,C 180,E1 13160.037,E2 13160.037} C_VEL
LIN {X 0,Y 392.253,Z 975.743,A -85,B 0,C 180,E1 13158.968,E2 13158.968} C_VEL
LIN {X 0,Y 401.636,Z 946.196,A -85,B 0,C 180,E1 13157.831,E2 13157.831} C_VEL
LIN {X 0,Y 408.04,Z 922.752,A -85,B 0,C 180,E1 13157.124,E2 13157.124} C_VEL
LIN {X 0,Y 413.836,Z 897.303,A -85,B 0,C 180,E1 13156.475,E2 13156.475} C_VEL
LIN {X 0,Y 418.817,Z 867.733,A -85,B 0,C 180,E1 13155.838,E2 13155.838} C_VEL
LIN {X 0,Y 446.639,Z 639.037,A -85,B 0,C 180,E1 13151.872,E2 13151.872} C_VEL
LIN {X 0,Y 449.394,Z 616.854,A -85,B 0,C 180,E1 13151.486,E2 13151.486} C_VEL
LIN {X 0,Y 441.669,Z 603.586,A -85,B 0,C 180,E1 13148.265,E2 13148.265} C_VEL
LIN {X 0,Y 434.231,Z 591.312,A -85,B 0,C 180,E1 13144.788,E2 13144.788} C_VEL
LIN {X 0,Y 427.242,Z 580.204,A -85,B 0,C 180,E1 13141.073,E2 13141.073} C_VEL
LIN {X 0,Y 421.892,Z 572.05,A -85,B 0,C 180,E1 13137.827,E2 13137.827} C_VEL
LIN {X 0,Y 416.725,Z 564.157,A -85,B 0,C 180,E1 13134.216,E2 13134.216} C_VEL
LIN {X 0,Y 413.62,Z 559.524,A -85,B 0,C 180,E1 13131.73,E2 13131.73} C_VEL
LIN {X 0,Y 410.358,Z 554.534,A -85,B 0,C 180,E1 13128.759,E2 13128.759} C_VEL
LIN {X 0,Y 407.151,Z 549.533,A -85,B 0,C 180,E1 13125.348,E2 13125.348} C_VEL
LIN {X 0,Y 404.377,Z 545.553,A -85,B 0,C 180,E1 13121.847,E2 13121.847} C_VEL
LIN {X 0,Y 401.965,Z 543.546,A -85,B 0,C 180,E1 13118.398,E2 13118.398} C_VEL
LIN {X 0,Y 400.281,Z 540.585,A -85,B 0,C 180,E1 13114.713,E2 13114.713} C_VEL
LIN {X 0,Y 399.709,Z 539.609,A -85,B 0,C 180,E1 13113.078,E2 13113.078} C_VEL
LIN {X 0,Y 398.394,Z 539.002,A -85,B 0,C 180,E1 13108.851,E2 13108.851} C_VEL
LIN {X 0,Y 398.032,Z 538.683,A -85,B 0,C 180,E1 13104.352,E2 13104.352} C_VEL
LIN {X 0,Y 398.494,Z 538.96,A -85,B 0,C 180,E1 13099.656,E2 13099.656} C_VEL
LIN {X 0,Y 400.029,Z 539.664,A -85,B 0,C 180,E1 13095.18,E2 13095.18} C_VEL
LIN {X 0,Y 400.576,Z 540.424,A -85,B 0,C 180,E1 13093.831,E2 13093.831} C_VEL
LIN {X 0,Y 402.755,Z 543.97,A -85,B 0,C 180,E1 13089.645,E2 13089.645} C_VEL
LIN {X 0,Y 405.49,Z 546.217,A -85,B 0,C 180,E1 13086.206,E2 13086.206} C_VEL
LIN {X 0,Y 408.47,Z 550.391,A -85,B 0,C 180,E1 13082.899,E2 13082.899} C_VEL
LIN {X 0,Y 410.43,Z 552.298,A -85,B 0,C 180,E1 13081.152,E2 13081.152} C_VEL
LIN {X 0,Y 414.328,Z 557.06,A -85,B 0,C 180,E1 13077.961,E2 13077.961} C_VEL
LIN {X 0,Y 419.59,Z 563.871,A -85,B 0,C 180,E1 13074.272,E2 13074.272} C_VEL
LIN {X 0,Y 424.004,Z 569.591,A -85,B 0,C 180,E1 13071.626,E2 13071.626} C_VEL
LIN {X 0,Y 428.732,Z 575.818,A -85,B 0,C 180,E1 13069.057,E2 13069.057} C_VEL
LIN {X 0,Y 435.447,Z 585.052,A -85,B 0,C 180,E1 13065.818,E2 13065.818} C_VEL
LIN {X 0,Y 443.501,Z 596.453,A -85,B 0,C 180,E1 13062.409,E2 13062.409} C_VEL
LIN {X 0,Y 445.092,Z 599.047,A -85,B 0,C 180,E1 13061.769,E2 13061.769} C_VEL
LIN {X 0,Y 421.174,Z 795.617,A -85,B 0,C 180,E1 13058.407,E2 13058.407} C_VEL
LIN {X 0,Y 416.074,Z 826.238,A -85,B 0,C 180,E1 13057.682,E2 13057.682} C_VEL
LIN {X 0,Y 410.975,Z 850.34,A -85,B 0,C 180,E1 13056.947,E2 13056.947} C_VEL
LIN {X 0,Y 404.343,Z 876.837,A -85,B 0,C 180,E1 13055.961,E2 13055.961} C_VEL
LIN {X 0,Y 396.311,Z 903.449,A -85,B 0,C 180,E1 13054.735,E2 13054.735} C_VEL
LIN {X 0,Y 388.88,Z 925.245,A -85,B 0,C 180,E1 13053.538,E2 13053.538} C_VEL
LIN {X 0,Y 379.605,Z 949.641,A -85,B 0,C 180,E1 13051.962,E2 13051.962} C_VEL
LIN {X 0,Y 369.965,Z 971.969,A -85,B 0,C 180,E1 13050.231,E2 13050.231} C_VEL
LIN {X 0,Y 361.082,Z 990.91,A -85,B 0,C 180,E1 13048.523,E2 13048.523} C_VEL
LIN {X 0,Y 351.304,Z 1010.295,A -85,B 0,C 180,E1 13046.492,E2 13046.492} C_VEL
LIN {X 0,Y 339.289,Z 1032.206,A -85,B 0,C 180,E1 13043.74,E2 13043.74} C_VEL
LIN {X 0,Y 329.56,Z 1048.678,A -85,B 0,C 180,E1 13041.275,E2 13041.275} C_VEL
LIN {X 0,Y 319.953,Z 1064.187,A -85,B 0,C 180,E1 13038.563,E2 13038.563} C_VEL
LIN {X 0,Y 308.156,Z 1082.316,A -85,B 0,C 180,E1 13034.763,E2 13034.763} C_VEL
LIN {X 0,Y 299.181,Z 1095.545,A -85,B 0,C 180,E1 13031.41,E2 13031.41} C_VEL
LIN {X 0,Y 291.779,Z 1106.284,A -85,B 0,C 180,E1 13028.231,E2 13028.231} C_VEL
LIN {X 0,Y 284.742,Z 1116.439,A -85,B 0,C 180,E1 13024.727,E2 13024.727} C_VEL
LIN {X 0,Y 277.812,Z 1126.622,A -85,B 0,C 180,E1 13020.575,E2 13020.575} C_VEL
LIN {X 0,Y 270.642,Z 1137.493,A -85,B 0,C 180,E1 13015.103,E2 13015.103} C_VEL
LIN {X 0,Y 266.234,Z 1144.701,A -85,B 0,C 180,E1 13010.602,E2 13010.602} C_VEL
LIN {X 0,Y 263.05,Z 1150.494,A -85,B 0,C 180,E1 13006.228,E2 13006.228} C_VEL
LIN {X 0,Y 260.759,Z 1155.514,A -85,B 0,C 180,E1 13001.558,E2 13001.558} C_VEL
LIN {X 0,Y 259.223,Z 1160.228,A -85,B 0,C 180,E1 12995.895,E2 12995.895} C_VEL
LIN {X 0,Y 258.646,Z 1163.186,A -85,B 0,C 180,E1 12990.684,E2 12990.684} C_VEL
LIN {X 0,Y 258.586,Z 1164.923,A -85,B 0,C 180,E1 12986.156,E2 12986.156} C_VEL
LIN {X 0,Y 258.792,Z 1165.851,A -85,B 0,C 180,E1 12981.987,E2 12981.987} C_VEL
LIN {X 0,Y 259.369,Z 1166.133,A -85,B 0,C 180,E1 12977.731,E2 12977.731} C_VEL
LIN {X 0,Y 260.512,Z 1165.661,A -85,B 0,C 180,E1 12973.088,E2 12973.088} C_VEL
LIN {X 0,Y 262.521,Z 1164.347,A -85,B 0,C 180,E1 12968.322,E2 12968.322} C_VEL
LIN {X 0,Y 265.729,Z 1162.094,A -85,B 0,C 180,E1 12963.452,E2 12963.452} C_VEL
LIN {X 0,Y 271.657,Z 1157.955,A -85,B 0,C 180,E1 12957.506,E2 12957.506} C_VEL
LIN {X 0,Y 272.663,Z 1156.856,A -85,B 0,C 180,E1 12955.903,E2 12955.903} C_VEL
LIN {X 0,Y 273.052,Z 1154.809,A -85,B 0,C 180,E1 12951.46,E2 12951.46} C_VEL
LIN {X 0,Y 274.623,Z 1153.642,A -85,B 0,C 180,E1 12950.127,E2 12950.127} C_VEL
LIN {X 0,Y 287.035,Z 1145.865,A -85,B 0,C 180,E1 12944.234,E2 12944.234} C_VEL
LIN {X 0,Y 302.775,Z 1136.283,A -85,B 0,C 180,E1 12938.699,E2 12938.699} C_VEL
LIN {X 0,Y 325.805,Z 1122.586,A -85,B 0,C 180,E1 12932.788,E2 12932.788} C_VEL
LIN {X 0,Y 331.034,Z 1119.514,A -85,B 0,C 180,E1 12931.691,E2 12931.691} C_VEL
LIN {X 0,Y 308.626,Z 1142.762,A -85,B 0,C 180,E1 12926.705,E2 12926.705} C_VEL
LIN {X 0,Y 288.006,Z 1168.114,A -85,B 0,C 180,E1 12920.107,E2 12920.107} C_VEL
LIN {X 0,Y 276.653,Z 1184.065,A -85,B 0,C 180,E1 12915.103,E2 12915.103} C_VEL
LIN {X 0,Y 268.067,Z 1197.427,A -85,B 0,C 180,E1 12910.187,E2 12910.187} C_VEL
LIN {X 0,Y 260.307,Z 1211.333,A -85,B 0,C 180,E1 12904.111,E2 12904.111} C_VEL
LIN {X 0,Y 255.244,Z 1222.119,A -85,B 0,C 180,E1 12898.294,E2 12898.294} C_VEL
LIN {X 0,Y 252.444,Z 1229.933,A -85,B 0,C 180,E1 12893.232,E2 12893.232} C_VEL
LIN {X 0,Y 250.928,Z 1235.869,A -85,B 0,C 180,E1 12888.589,E2 12888.589} C_VEL
LIN {X 0,Y 250.326,Z 1240.318,A -85,B 0,C 180,E1 12884.338,E2 12884.338} C_VEL
LIN {X 0,Y 250.292,Z 1243.94,A -85,B 0,C 180,E1 12879.891,E2 12879.891} C_VEL
LIN {X 0,Y 250.55,Z 1246.404,A -85,B 0,C 180,E1 12875.496,E2 12875.496} C_VEL
LIN {X 0,Y 250.7,Z 1247.663,A -85,B 0,C 180,E1 12871.371,E2 12871.371} C_VEL
LIN {X 0,Y 250.598,Z 1247.777,A -85,B 0,C 180,E1 12867.027,E2 12867.027} C_VEL
LIN {X 0,Y 250.245,Z 1246.657,A -85,B 0,C 180,E1 12862.654,E2 12862.654} C_VEL
LIN {X 0,Y 250.061,Z 1244.022,A -85,B 0,C 180,E1 12857.765,E2 12857.765} C_VEL
LIN {X 0,Y 250.445,Z 1240.225,A -85,B 0,C 180,E1 12853.055,E2 12853.055} C_VEL
LIN {X 0,Y 251.632,Z 1235.278,A -85,B 0,C 180,E1 12848.409,E2 12848.409} C_VEL
LIN {X 0,Y 253.759,Z 1229.376,A -85,B 0,C 180,E1 12843.948,E2 12843.948} C_VEL
LIN {X 0,Y 256.878,Z 1222.445,A -85,B 0,C 180,E1 12839.601,E2 12839.601} C_VEL
LIN {X 0,Y 261.467,Z 1213.686,A -85,B 0,C 180,E1 12834.997,E2 12834.997} C_VEL
LIN {X 0,Y 268.684,Z 1201.339,A -85,B 0,C 180,E1 12829.645,E2 12829.645} C_VEL
LIN {X 0,Y 276.767,Z 1188.317,A -85,B 0,C 180,E1 12825.081,E2 12825.081} C_VEL
LIN {X 0,Y 284.431,Z 1176.284,A -85,B 0,C 180,E1 12821.516,E2 12821.516} C_VEL
LIN {X 0,Y 293.791,Z 1161.691,A -85,B 0,C 180,E1 12817.854,E2 12817.854} C_VEL
LIN {X 0,Y 305.354,Z 1143.345,A -85,B 0,C 180,E1 12814.052,E2 12814.052} C_VEL
LIN {X 0,Y 315.56,Z 1126.663,A -85,B 0,C 180,E1 12811.183,E2 12811.183} C_VEL
LIN {X 0,Y 325.506,Z 1109.829,A -85,B 0,C 180,E1 12808.719,E2 12808.719} C_VEL
LIN {X 0,Y 337.786,Z 1088.016,A -85,B 0,C 180,E1 12806.041,E2 12806.041} C_VEL
LIN {X 0,Y 348.874,Z 1066.764,A -85,B 0,C 180,E1 12803.9,E2 12803.9} C_VEL
LIN {X 0,Y 358.159,Z 1047.814,A -85,B 0,C 180,E1 12802.285,E2 12802.285} C_VEL
LIN {X 0,Y 368.983,Z 1024.028,A -85,B 0,C 180,E1 12800.571,E2 12800.571} C_VEL
LIN {X 0,Y 379.184,Z 998.921,A -85,B 0,C 180,E1 12799.109,E2 12799.109} C_VEL
LIN {X 0,Y 387.067,Z 977.637,A -85,B 0,C 180,E1 12798.081,E2 12798.081} C_VEL
LIN {X 0,Y 395.4,Z 952.686,A -85,B 0,C 180,E1 12797.084,E2 12797.084} C_VEL
LIN {X 0,Y 403.26,Z 925.099,A -85,B 0,C 180,E1 12796.224,E2 12796.224} C_VEL
LIN {X 0,Y 408.809,Z 901.827,A -85,B 0,C 180,E1 12795.625,E2 12795.625} C_VEL
LIN {X 0,Y 414.023,Z 874.167,A -85,B 0,C 180,E1 12794.998,E2 12794.998} C_VEL
LIN {X 0,Y 420.09,Z 826.817,A -85,B 0,C 180,E1 12794.135,E2 12794.135} C_VEL
LIN {X 0,Y 445.649,Z 621.833,A -85,B 0,C 180,E1 12790.631,E2 12790.631} C_VEL
LIN {X 0,Y 439.236,Z 610.624,A -85,B 0,C 180,E1 12787.883,E2 12787.883} C_VEL
LIN {X 0,Y 432.134,Z 598.755,A -85,B 0,C 180,E1 12784.512,E2 12784.512} C_VEL
LIN {X 0,Y 424.923,Z 587.153,A -85,B 0,C 180,E1 12780.613,E2 12780.613} C_VEL
LIN {X 0,Y 418.663,Z 577.361,A -85,B 0,C 180,E1 12776.65,E2 12776.65} C_VEL
LIN {X 0,Y 413.645,Z 569.735,A -85,B 0,C 180,E1 12772.918,E2 12772.918} C_VEL
LIN {X 0,Y 408.786,Z 562.418,A -85,B 0,C 180,E1 12768.715,E2 12768.715} C_VEL
LIN {X 0,Y 405.427,Z 557.225,A -85,B 0,C 180,E1 12765.138,E2 12765.138} C_VEL
LIN {X 0,Y 402.791,Z 553.378,A -85,B 0,C 180,E1 12761.773,E2 12761.773} C_VEL
LIN {X 0,Y 400.366,Z 551.345,A -85,B 0,C 180,E1 12758.285,E2 12758.285} C_VEL
LIN {X 0,Y 398.609,Z 548.04,A -85,B 0,C 180,E1 12754.226,E2 12754.226} C_VEL
LIN {X 0,Y 397.559,Z 547.195,A -85,B 0,C 180,E1 12751.454,E2 12751.454} C_VEL
LIN {X 0,Y 396.509,Z 546.605,A -85,B 0,C 180,E1 12746.321,E2 12746.321} C_VEL
LIN {X 0,Y 396.544,Z 546.606,A -85,B 0,C 180,E1 12742.213,E2 12742.213} C_VEL
LIN {X 0,Y 397.683,Z 547.16,A -85,B 0,C 180,E1 12737.236,E2 12737.236} C_VEL
LIN {X 0,Y 398.951,Z 547.991,A -85,B 0,C 180,E1 12734.166,E2 12734.166} C_VEL
LIN {X 0,Y 400.98,Z 551.568,A -85,B 0,C 180,E1 12730.042,E2 12730.042} C_VEL
LIN {X 0,Y 403.838,Z 553.955,A -85,B 0,C 180,E1 12726.378,E2 12726.378} C_VEL
LIN {X 0,Y 406.808,Z 558.141,A -85,B 0,C 180,E1 12723.055,E2 12723.055} C_VEL
LIN {X 0,Y 408.77,Z 560.05,A -85,B 0,C 180,E1 12721.318,E2 12721.318} C_VEL
LIN {X 0,Y 413.274,Z 565.795,A -85,B 0,C 180,E1 12717.609,E2 12717.609} C_VEL
LIN {X 0,Y 417.782,Z 571.486,A -85,B 0,C 180,E1 12714.501,E2 12714.501} C_VEL
LIN {X 0,Y 422.192,Z 577.283,A -85,B 0,C 180,E1 12711.815,E2 12711.815} C_VEL
LIN {X 0,Y 426.849,Z 583.461,A -85,B 0,C 180,E1 12709.26,E2 12709.26} C_VEL
LIN {X 0,Y 433.398,Z 592.554,A -85,B 0,C 180,E1 12706.072,E2 12706.072} C_VEL
LIN {X 0,Y 441.191,Z 603.7,A -85,B 0,C 180,E1 12702.733,E2 12702.733} C_VEL
LIN {X 0,Y 441.367,Z 604.339,A -85,B 0,C 180,E1 12702.64,E2 12702.64} C_VEL
LIN {X 0,Y 417.549,Z 795.857,A -85,B 0,C 180,E1 12699.382,E2 12699.382} C_VEL
LIN {X 0,Y 412.362,Z 826.617,A -85,B 0,C 180,E1 12698.661,E2 12698.661} C_VEL
LIN {X 0,Y 407.221,Z 850.601,A -85,B 0,C 180,E1 12697.939,E2 12697.939} C_VEL
LIN {X 0,Y 400.871,Z 875.692,A -85,B 0,C 180,E1 12697.02,E2 12697.02} C_VEL
LIN {X 0,Y 392.693,Z 902.765,A -85,B 0,C 180,E1 12695.8,E2 12695.8} C_VEL
LIN {X 0,Y 385.139,Z 924.651,A -85,B 0,C 180,E1 12694.616,E2 12694.616} C_VEL
LIN {X 0,Y 376.917,Z 946.046,A -85,B 0,C 180,E1 12693.269,E2 12693.269} C_VEL
LIN {X 0,Y 366.067,Z 971.243,A -85,B 0,C 180,E1 12691.375,E2 12691.375} C_VEL
LIN {X 0,Y 356.969,Z 990.349,A -85,B 0,C 180,E1 12689.676,E2 12689.676} C_VEL
LIN {X 0,Y 347.454,Z 1008.91,A -85,B 0,C 180,E1 12687.76,E2 12687.76} C_VEL
LIN {X 0,Y 335.972,Z 1029.78,A -85,B 0,C 180,E1 12685.22,E2 12685.22} C_VEL
LIN {X 0,Y 324.764,Z 1048.448,A -85,B 0,C 180,E1 12682.474,E2 12682.474} C_VEL
LIN {X 0,Y 315.58,Z 1063.012,A -85,B 0,C 180,E1 12679.964,E2 12679.964} C_VEL
LIN {X 0,Y 305.746,Z 1077.954,A -85,B 0,C 180,E1 12676.959,E2 12676.959} C_VEL
LIN {X 0,Y 293.994,Z 1094.996,A -85,B 0,C 180,E1 12672.789,E2 12672.789} C_VEL
LIN {X 0,Y 285.489,Z 1106.952,A -85,B 0,C 180,E1 12669.251,E2 12669.251} C_VEL
LIN {X 0,Y 278.136,Z 1117.218,A -85,B 0,C 180,E1 12665.677,E2 12665.677} C_VEL
LIN {X 0,Y 271.336,Z 1126.826,A -85,B 0,C 180,E1 12661.731,E2 12661.731} C_VEL
LIN {X 0,Y 264.066,Z 1137.503,A -85,B 0,C 180,E1 12656.412,E2 12656.412} C_VEL
LIN {X 0,Y 259.07,Z 1145.233,A -85,B 0,C 180,E1 12651.581,E2 12651.581} C_VEL
LIN {X 0,Y 255.593,Z 1151.247,A -85,B 0,C 180,E1 12647.017,E2 12647.017} C_VEL
LIN {X 0,Y 253.346,Z 1155.854,A -85,B 0,C 180,E1 12642.753,E2 12642.753} C_VEL
LIN {X 0,Y 251.784,Z 1159.764,A -85,B 0,C 180,E1 12638.281,E2 12638.281} C_VEL
LIN {X 0,Y 251.009,Z 1162.591,A -85,B 0,C 180,E1 12634.172,E2 12634.172} C_VEL
LIN {X 0,Y 250.716,Z 1164.743,A -85,B 0,C 180,E1 12630.071,E2 12630.071} C_VEL
LIN {X 0,Y 250.708,Z 1166.376,A -85,B 0,C 180,E1 12625.666,E2 12625.666} C_VEL
LIN {X 0,Y 251.021,Z 1167.32,A -85,B 0,C 180,E1 12621.239,E2 12621.239} C_VEL
LIN {X 0,Y 251.686,Z 1167.578,A -85,B 0,C 180,E1 12616.78,E2 12616.78} C_VEL
LIN {X 0,Y 252.98,Z 1167.13,A -85,B 0,C 180,E1 12612.092,E2 12612.092} C_VEL
LIN {X 0,Y 255.465,Z 1165.745,A -85,B 0,C 180,E1 12606.969,E2 12606.969} C_VEL
LIN {X 0,Y 260.564,Z 1162.573,A -85,B 0,C 180,E1 12600.44,E2 12600.44} C_VEL
LIN {X 0,Y 267.011,Z 1158.423,A -85,B 0,C 180,E1 12594.93,E2 12594.93} C_VEL
LIN {X 0,Y 274.623,Z 1153.642,A -85,B 0,C 180,E1 12590.127,E2 12590.127} C_VEL
LIN {X 0,Y 276.628,Z 1152.268,A -85,B 0,C 180,E1 12588.472,E2 12588.472} C_VEL
LIN {X 0,Y 279.494,Z 1149.732,A -85,B 0,C 180,E1 12584.283,E2 12584.283} C_VEL
LIN {X 0,Y 281.757,Z 1148.3,A -85,B 0,C 180,E1 12583.039,E2 12583.039} C_VEL
LIN {X 0,Y 299.883,Z 1138.204,A -85,B 0,C 180,E1 12577.039,E2 12577.039} C_VEL
LIN {X 0,Y 321.431,Z 1126.629,A -85,B 0,C 180,E1 12571.803,E2 12571.803} C_VEL
LIN {X 0,Y 300.343,Z 1147.334,A -85,B 0,C 180,E1 12567.028,E2 12567.028} C_VEL
LIN {X 0,Y 278.531,Z 1172.91,A -85,B 0,C 180,E1 12559.874,E2 12559.874} C_VEL
LIN {X 0,Y 265.261,Z 1190.815,A -85,B 0,C 180,E1 12553.614,E2 12553.614} C_VEL
LIN {X 0,Y 257.567,Z 1202.667,A -85,B 0,C 180,E1 12548.682,E2 12548.682} C_VEL
LIN {X 0,Y 251.75,Z 1212.74,A -85,B 0,C 180,E1 12543.782,E2 12543.782} C_VEL
LIN {X 0,Y 247.636,Z 1221.168,A -85,B 0,C 180,E1 12538.981,E2 12538.981} C_VEL
LIN {X 0,Y 244.795,Z 1228.429,A -85,B 0,C 180,E1 12534.108,E2 12534.108} C_VEL
LIN {X 0,Y 243.163,Z 1234.234,A -85,B 0,C 180,E1 12529.455,E2 12529.455} C_VEL
LIN {X 0,Y 242.426,Z 1238.943,A -85,B 0,C 180,E1 12524.816,E2 12524.816} C_VEL
LIN {X 0,Y 242.363,Z 1242.553,A -85,B 0,C 180,E1 12520.218,E2 12520.218} C_VEL
LIN {X 0,Y 242.637,Z 1245.04,A -85,B 0,C 180,E1 12515.676,E2 12515.676} C_VEL
LIN {X 0,Y 242.819,Z 1246.289,A -85,B 0,C 180,E1 12511.416,E2 12511.416} C_VEL
LIN {X 0,Y 242.723,Z 1246.421,A -85,B 0,C 180,E1 12507.166,E2 12507.166} C_VEL
LIN {X 0,Y 242.351,Z 1245.327,A -85,B 0,C 180,E1 12502.652,E2 12502.652} C_VEL
LIN {X 0,Y 242.151,Z 1242.702,A -85,B 0,C 180,E1 12497.601,E2 12497.601} C_VEL
LIN {X 0,Y 242.564,Z 1238.907,A -85,B 0,C 180,E1 12492.735,E2 12492.735} C_VEL
LIN {X 0,Y 243.774,Z 1234.131,A -85,B 0,C 180,E1 12488.084,E2 12488.084} C_VEL
LIN {X 0,Y 245.876,Z 1228.553,A -85,B 0,C 180,E1 12483.688,E2 12483.688} C_VEL
LIN {X 0,Y 249.179,Z 1221.514,A -85,B 0,C 180,E1 12479.094,E2 12479.094} C_VEL
LIN {X 0,Y 253.688,Z 1213.265,A -85,B 0,C 180,E1 12474.593,E2 12474.593} C_VEL
LIN {X 0,Y 260.076,Z 1202.684,A -85,B 0,C 180,E1 12469.768,E2 12469.768} C_VEL
LIN {X 0,Y 269.224,Z 1188.429,A -85,B 0,C 180,E1 12464.515,E2 12464.515} C_VEL
LIN {X 0,Y 277.435,Z 1175.954,A -85,B 0,C 180,E1 12460.718,E2 12460.718} C_VEL
LIN {X 0,Y 286.759,Z 1161.894,A -85,B 0,C 180,E1 12457.102,E2 12457.102} C_VEL
LIN {X 0,Y 298.736,Z 1143.582,A -85,B 0,C 180,E1 12453.201,E2 12453.201} C_VEL
LIN {X 0,Y 309.833,Z 1125.961,A -85,B 0,C 180,E1 12450.132,E2 12450.132} C_VEL
LIN {X 0,Y 319.694,Z 1109.699,A -85,B 0,C 180,E1 12447.735,E2 12447.735} C_VEL
LIN {X 0,Y 331.748,Z 1088.887,A -85,B 0,C 180,E1 12445.149,E2 12445.149} C_VEL
LIN {X 0,Y 343.555,Z 1066.753,A -85,B 0,C 180,E1 12442.907,E2 12442.907} C_VEL
LIN {X 0,Y 353.385,Z 1047.1,A -85,B 0,C 180,E1 12441.234,E2 12441.234} C_VEL
LIN {X 0,Y 364.136,Z 1023.971,A -85,B 0,C 180,E1 12439.573,E2 12439.573} C_VEL
LIN {X 0,Y 374.527,Z 999.025,A -85,B 0,C 180,E1 12438.119,E2 12438.119} C_VEL
LIN {X 0,Y 382.393,Z 978.266,A -85,B 0,C 180,E1 12437.117,E2 12437.117} C_VEL
LIN {X 0,Y 390.17,Z 955.551,A -85,B 0,C 180,E1 12436.204,E2 12436.204} C_VEL
LIN {X 0,Y 399.047,Z 925.576,A -85,B 0,C 180,E1 12435.254,E2 12435.254} C_VEL
LIN {X 0,Y 404.798,Z 902.034,A -85,B 0,C 180,E1 12434.651,E2 12434.651} C_VEL
LIN {X 0,Y 409.616,Z 877.341,A -85,B 0,C 180,E1 12434.09,E2 12434.09} C_VEL
LIN {X 0,Y 414.763,Z 840.437,A -85,B 0,C 180,E1 12433.396,E2 12433.396} C_VEL
LIN {X 0,Y 442.001,Z 626.737,A -85,B 0,C 180,E1 12429.76,E2 12429.76} C_VEL
LIN {X 0,Y 434.775,Z 614.123,A -85,B 0,C 180,E1 12426.539,E2 12426.539} C_VEL
LIN {X 0,Y 427.855,Z 602.612,A -85,B 0,C 180,E1 12423.081,E2 12423.081} C_VEL
LIN {X 0,Y 422.257,Z 593.654,A -85,B 0,C 180,E1 12419.932,E2 12419.932} C_VEL
LIN {X 0,Y 416.657,Z 584.707,A -85,B 0,C 180,E1 12416.285,E2 12416.285} C_VEL
LIN {X 0,Y 411.504,Z 576.883,A -85,B 0,C 180,E1 12412.46,E2 12412.46} C_VEL
LIN {X 0,Y 406.886,Z 569.916,A -85,B 0,C 180,E1 12408.375,E2 12408.375} C_VEL
LIN {X 0,Y 403.708,Z 564.916,A -85,B 0,C 180,E1 12404.926,E2 12404.926} C_VEL
LIN {X 0,Y 401.206,Z 561.204,A -85,B 0,C 180,E1 12401.698,E2 12401.698} C_VEL
LIN {X 0,Y 398.707,Z 559.058,A -85,B 0,C 180,E1 12398.058,E2 12398.058} C_VEL
LIN {X 0,Y 396.747,Z 555.423,A -85,B 0,C 180,E1 12393.346,E2 12393.346} C_VEL
LIN {X 0,Y 395.333,Z 554.708,A -85,B 0,C 180,E1 12388.938,E2 12388.938} C_VEL
LIN {X 0,Y 394.936,Z 554.388,A -85,B 0,C 180,E1 12384.565,E2 12384.565} C_VEL
LIN {X 0,Y 395.405,Z 554.65,A -85,B 0,C 180,E1 12379.79,E2 12379.79} C_VEL
LIN {X 0,Y 396.948,Z 555.356,A -85,B 0,C 180,E1 12375.262,E2 12375.262} C_VEL
LIN {X 0,Y 397.441,Z 556.021,A -85,B 0,C 180,E1 12374.088,E2 12374.088} C_VEL
LIN {X 0,Y 399.757,Z 559.755,A -85,B 0,C 180,E1 12369.611,E2 12369.611} C_VEL
LIN {X 0,Y 402.267,Z 561.851,A -85,B 0,C 180,E1 12366.446,E2 12366.446} C_VEL
LIN {X 0,Y 405.149,Z 565.891,A -85,B 0,C 180,E1 12363.213,E2 12363.213} C_VEL
LIN {X 0,Y 407.064,Z 567.719,A -85,B 0,C 180,E1 12361.531,E2 12361.531} C_VEL
LIN {X 0,Y 411.552,Z 573.488,A -85,B 0,C 180,E1 12357.805,E2 12357.805} C_VEL
LIN {X 0,Y 416.078,Z 579.278,A -85,B 0,C 180,E1 12354.649,E2 12354.649} C_VEL
LIN {X 0,Y 420.303,Z 584.889,A -85,B 0,C 180,E1 12352.038,E2 12352.038} C_VEL
LIN {X 0,Y 424.861,Z 590.96,A -85,B 0,C 180,E1 12349.523,E2 12349.523} C_VEL
LIN {X 0,Y 431.535,Z 600.297,A -85,B 0,C 180,E1 12346.247,E2 12346.247} C_VEL
LIN {X 0,Y 437.759,Z 609.298,A -85,B 0,C 180,E1 12343.531,E2 12343.531} C_VEL
LIN {X 0,Y 413.72,Z 797.797,A -85,B 0,C 180,E1 12340.334,E2 12340.334} C_VEL
LIN {X 0,Y 408.41,Z 828.305,A -85,B 0,C 180,E1 12339.616,E2 12339.616} C_VEL
LIN {X 0,Y 403.078,Z 852.601,A -85,B 0,C 180,E1 12338.883,E2 12338.883} C_VEL
LIN {X 0,Y 395.96,Z 879.909,A -85,B 0,C 180,E1 12337.874,E2 12337.874} C_VEL
LIN {X 0,Y 388.007,Z 905.284,A -85,B 0,C 180,E1 12336.715,E2 12336.715} C_VEL
LIN {X 0,Y 380.162,Z 927.516,A -85,B 0,C 180,E1 12335.509,E2 12335.509} C_VEL
LIN {X 0,Y 370.534,Z 951.913,A -85,B 0,C 180,E1 12333.946,E2 12333.946} C_VEL
LIN {X 0,Y 360.523,Z 974.281,A -85,B 0,C 180,E1 12332.225,E2 12332.225} C_VEL
LIN {X 0,Y 351.381,Z 993.018,A -85,B 0,C 180,E1 12330.544,E2 12330.544} C_VEL
LIN {X 0,Y 340.763,Z 1013.19,A -85,B 0,C 180,E1 12328.428,E2 12328.428} C_VEL
LIN {X 0,Y 328.844,Z 1033.916,A -85,B 0,C 180,E1 12325.813,E2 12325.813} C_VEL
LIN {X 0,Y 319.055,Z 1049.819,A -85,B 0,C 180,E1 12323.441,E2 12323.441} C_VEL
LIN {X 0,Y 309.567,Z 1064.484,A -85,B 0,C 180,E1 12320.894,E2 12320.894} C_VEL
LIN {X 0,Y 299.474,Z 1079.424,A -85,B 0,C 180,E1 12317.858,E2 12317.858} C_VEL
LIN {X 0,Y 287.545,Z 1096.279,A -85,B 0,C 180,E1 12313.689,E2 12313.689} C_VEL
LIN {X 0,Y 278.734,Z 1108.335,A -85,B 0,C 180,E1 12310.075,E2 12310.075} C_VEL
LIN {X 0,Y 270.833,Z 1119.057,A -85,B 0,C 180,E1 12306.271,E2 12306.271} C_VEL
LIN {X 0,Y 262.455,Z 1130.65,A -85,B 0,C 180,E1 12301.313,E2 12301.313} C_VEL
LIN {X 0,Y 255.518,Z 1140.368,A -85,B 0,C 180,E1 12296.058,E2 12296.058} C_VEL
LIN {X 0,Y 251.049,Z 1147.188,A -85,B 0,C 180,E1 12291.588,E2 12291.588} C_VEL
LIN {X 0,Y 247.591,Z 1153.036,A -85,B 0,C 180,E1 12286.961,E2 12286.961} C_VEL
LIN {X 0,Y 245.091,Z 1158.126,A -85,B 0,C 180,E1 12281.995,E2 12281.995} C_VEL
LIN {X 0,Y 243.375,Z 1163.044,A -85,B 0,C 180,E1 12275.69,E2 12275.69} C_VEL
LIN {X 0,Y 242.842,Z 1165.912,A -85,B 0,C 180,E1 12270.428,E2 12270.428} C_VEL
LIN {X 0,Y 242.819,Z 1167.713,A -85,B 0,C 180,E1 12265.605,E2 12265.605} C_VEL
LIN {X 0,Y 243.164,Z 1168.73,A -85,B 0,C 180,E1 12260.962,E2 12260.962} C_VEL
LIN {X 0,Y 243.899,Z 1169.078,A -85,B 0,C 180,E1 12256.404,E2 12256.404} C_VEL
LIN {X 0,Y 245.236,Z 1168.735,A -85,B 0,C 180,E1 12251.763,E2 12251.763} C_VEL
LIN {X 0,Y 247.747,Z 1167.557,A -85,B 0,C 180,E1 12246.721,E2 12246.721} C_VEL
LIN {X 0,Y 252.017,Z 1165.257,A -85,B 0,C 180,E1 12241.13,E2 12241.13} C_VEL
LIN {X 0,Y 259.67,Z 1160.881,A -85,B 0,C 180,E1 12234.476,E2 12234.476} C_VEL
LIN {X 0,Y 269.277,Z 1155.418,A -85,B 0,C 180,E1 12228.65,E2 12228.65} C_VEL
LIN {X 0,Y 281.757,Z 1148.3,A -85,B 0,C 180,E1 12223.039,E2 12223.039} C_VEL
LIN {X 0,Y 284.5,Z 1146.723,A -85,B 0,C 180,E1 12221.605,E2 12221.605} C_VEL
LIN {X 0,Y 289.997,Z 1143.908,A -85,B 0,C 180,E1 12217.668,E2 12217.668} C_VEL
LIN {X 0,Y 293.315,Z 1142.328,A -85,B 0,C 180,E1 12216.451,E2 12216.451} C_VEL
LIN {X 0,Y 311.794,Z 1133.18,A -85,B 0,C 180,E1 12211.954,E2 12211.954} C_VEL
LIN {X 0,Y 286.556,Z 1157.5,A -85,B 0,C 180,E1 12205.788,E2 12205.788} C_VEL
LIN {X 0,Y 268.079,Z 1178.425,A -85,B 0,C 180,E1 12199.213,E2 12199.213} C_VEL
LIN {X 0,Y 255.912,Z 1194.372,A -85,B 0,C 180,E1 12193.137,E2 12193.137} C_VEL
LIN {X 0,Y 246.289,Z 1208.825,A -85,B 0,C 180,E1 12186.351,E2 12186.351} C_VEL
LIN {X 0,Y 241,Z 1218.294,A -85,B 0,C 180,E1 12180.961,E2 12180.961} C_VEL
LIN {X 0,Y 237.523,Z 1226.079,A -85,B 0,C 180,E1 12175.695,E2 12175.695} C_VEL
LIN {X 0,Y 235.498,Z 1232.307,A -85,B 0,C 180,E1 12170.634,E2 12170.634} C_VEL
LIN {X 0,Y 234.59,Z 1237.147,A -85,B 0,C 180,E1 12165.83,E2 12165.83} C_VEL
